LIN {X 0,Y 675.364,Z 1023.131,A -85,B 0,C 180,E1 30768.288,E2 30768.288} C_VEL
LIN {X 0,Y 672.75,Z 1029.782,A -85,B 0,C 180,E1 30767.69,E2 30767.69} C_VEL
LIN {X 0,Y 672.369,Z 1032.5,A -85,B 0,C 180,E1 30767.398,E2 30767.398} C_VEL
LIN {X 0,Y 672.252,Z 1040.855,A -85,B 0,C 180,E1 30766.32,E2 30766.32} C_VEL
LIN {X 0,Y 672.157,Z 1047.422,A -85,B 0,C 180,E1 30765.175,E2 30765.175} C_VEL
LIN {X 0,Y 672.12,Z 1051.926,A -85,B 0,C 180,E1 30764.114,E2 30764.114} C_VEL
LIN {X 0,Y 672.089,Z 1055.278,A -85,B 0,C 180,E1 30762.957,E2 30762.957} C_VEL
LIN {X 0,Y 672.074,Z 1057.172,A -85,B 0,C 180,E1 30761.615,E2 30761.615} C_VEL
LIN {X 0,Y 672.069,Z 1057.276,A -85,B 0,C 180,E1 30760.533,E2 30760.533} C_VEL
LIN {X 0,Y 672.07,Z 1056.109,A -85,B 0,C 180,E1 30759.444,E2 30759.444} C_VEL
LIN {X 0,Y 672.096,Z 1053.112,A -85,B 0,C 180,E1 30758.165,E2 30758.165} C_VEL
LIN {X 0,Y 672.133,Z 1048.387,A -85,B 0,C 180,E1 30756.968,E2 30756.968} C_VEL
LIN {X 0,Y 672.186,Z 1042.857,A -85,B 0,C 180,E1 30755.947,E2 30755.947} C_VEL
LIN {X 0,Y 672.298,Z 1034.959,A -85,B 0,C 180,E1 30754.826,E2 30754.826} C_VEL
LIN {X 0,Y 672.444,Z 1025.328,A -85,B 0,C 180,E1 30753.792,E2 30753.792} C_VEL
LIN {X 0,Y 672.579,Z 1016.19,A -85,B 0,C 180,E1 30753.012,E2 30753.012} C_VEL
LIN {X 0,Y 672.716,Z 1005.111,A -85,B 0,C 180,E1 30752.247,E2 30752.247} C_VEL
LIN {X 0,Y 672.919,Z 991.221,A -85,B 0,C 180,E1 30751.512,E2 30751.512} C_VEL
LIN {X 0,Y 673.04,Z 978.297,A -85,B 0,C 180,E1 30751.008,E2 30751.008} C_VEL
LIN {X 0,Y 673.159,Z 964.07,A -85,B 0,C 180,E1 30750.609,E2 30750.609} C_VEL
LIN {X 0,Y 673.195,Z 947.441,A -85,B 0,C 180,E1 30750.341,E2 30750.341} C_VEL
LIN {X 0,Y 673.46,Z 838.836,A -85,B 0,C 180,E1 30749.163,E2 30749.163} C_VEL
LIN {X 0,Y 674.164,Z 758.895,A -85,B 0,C 180,E1 30746.003,E2 30746.003} C_VEL
LIN {X 0,Y 674.908,Z 679.946,A -85,B 0,C 180,E1 30742.883,E2 30742.883} C_VEL
LIN {X 0,Y 675.546,Z 603.018,A -85,B 0,C 180,E1 30739.85,E2 30739.85} C_VEL
LIN {X 0,Y 676.134,Z 525.625,A -85,B 0,C 180,E1 30736.788,E2 30736.788} C_VEL
LIN {X 0,Y 676.398,Z 479.441,A -85,B 0,C 180,E1 30734.947,E2 30734.947} C_VEL
LIN {X 0,Y 677.625,Z 481.415,A -85,B 0,C 180,E1 30734.815,E2 30734.815} C_VEL
LIN {X 0,Y 679.206,Z 481.602,A -85,B 0,C 180,E1 30734.68,E2 30734.68} C_VEL
LIN {X 0,Y 681.86,Z 479.707,A -85,B 0,C 180,E1 30734.487,E2 30734.487} C_VEL
LIN {X 0,Y 685.332,Z 474.609,A -85,B 0,C 180,E1 30734.275,E2 30734.275} C_VEL
LIN {X 0,Y 686.171,Z 473.174,A -85,B 0,C 180,E1 30734.227,E2 30734.227} C_VEL
LIN {X 0,Y 689.689,Z 471.896,A -85,B 0,C 180,E1 30733.961,E2 30733.961} C_VEL
LIN {X 0,Y 693.542,Z 468.674,A -85,B 0,C 180,E1 30733.699,E2 30733.699} C_VEL
LIN {X 0,Y 691.039,Z 679.216,A -85,B 0,C 180,E1 30730.991,E2 30730.991} C_VEL
LIN {X 0,Y 689.557,Z 799.238,A -85,B 0,C 180,E1 30729.461,E2 30729.461} C_VEL
LIN {X 0,Y 688.803,Z 826.662,A -85,B 0,C 180,E1 30728.964,E2 30728.964} C_VEL
LIN {X 0,Y 687.772,Z 853.657,A -85,B 0,C 180,E1 30728.297,E2 30728.297} C_VEL
LIN {X 0,Y 686.749,Z 876.496,A -85,B 0,C 180,E1 30727.594,E2 30727.594} C_VEL
LIN {X 0,Y 685.634,Z 898.908,A -85,B 0,C 180,E1 30726.779,E2 30726.779} C_VEL
LIN {X 0,Y 684.187,Z 925.781,A -85,B 0,C 180,E1 30725.624,E2 30725.624} C_VEL
LIN {X 0,Y 682.832,Z 948.662,A -85,B 0,C 180,E1 30724.47,E2 30724.47} C_VEL
LIN {X 0,Y 681.518,Z 969.977,A -85,B 0,C 180,E1 30723.25,E2 30723.25} C_VEL
LIN {X 0,Y 679.995,Z 993.701,A -85,B 0,C 180,E1 30721.715,E2 30721.715} C_VEL
LIN {X 0,Y 678.508,Z 1017.521,A -85,B 0,C 180,E1 30719.944,E2 30719.944} C_VEL
LIN {X 0,Y 677.131,Z 1039.319,A -85,B 0,C 180,E1 30718.103,E2 30718.103} C_VEL
LIN {X 0,Y 675.956,Z 1059.69,A -85,B 0,C 180,E1 30716.156,E2 30716.156} C_VEL
LIN {X 0,Y 674.879,Z 1078.449,A -85,B 0,C 180,E1 30714.124,E2 30714.124} C_VEL
LIN {X 0,Y 674.182,Z 1092.611,A -85,B 0,C 180,E1 30712.406,E2 30712.406} C_VEL
LIN {X 0,Y 673.586,Z 1105.407,A -85,B 0,C 180,E1 30710.69,E2 30710.69} C_VEL
LIN {X 0,Y 673.039,Z 1119.756,A -85,B 0,C 180,E1 30708.538,E2 30708.538} C_VEL
LIN {X 0,Y 672.594,Z 1131.955,A -85,B 0,C 180,E1 30706.408,E2 30706.408} C_VEL
LIN {X 0,Y 672.363,Z 1141.26,A -85,B 0,C 180,E1 30704.557,E2 30704.557} C_VEL
LIN {X 0,Y 672.181,Z 1149.32,A -85,B 0,C 180,E1 30702.719,E2 30702.719} C_VEL
LIN {X 0,Y 672.03,Z 1156.847,A -85,B 0,C 180,E1 30700.719,E2 30700.719} C_VEL
LIN {X 0,Y 671.972,Z 1163.694,A -85,B 0,C 180,E1 30698.472,E2 30698.472} C_VEL
LIN {X 0,Y 671.93,Z 1169.194,A -85,B 0,C 180,E1 30696.066,E2 30696.066} C_VEL
LIN {X 0,Y 671.912,Z 1172.615,A -85,B 0,C 180,E1 30693.841,E2 30693.841} C_VEL
LIN {X 0,Y 671.907,Z 1174.487,A -85,B 0,C 180,E1 30691.707,E2 30691.707} C_VEL
LIN {X 0,Y 671.892,Z 1174.892,A -85,B 0,C 180,E1 30689.404,E2 30689.404} C_VEL
LIN {X 0,Y 671.911,Z 1173.798,A -85,B 0,C 180,E1 30687.186,E2 30687.186} C_VEL
LIN {X 0,Y 671.921,Z 1170.978,A -85,B 0,C 180,E1 30684.879,E2 30684.879} C_VEL
LIN {X 0,Y 671.942,Z 1166.841,A -85,B 0,C 180,E1 30682.735,E2 30682.735} C_VEL
LIN {X 0,Y 671.993,Z 1161.255,A -85,B 0,C 180,E1 30680.58,E2 30680.58} C_VEL
LIN {X 0,Y 672.098,Z 1153.81,A -85,B 0,C 180,E1 30678.328,E2 30678.328} C_VEL
LIN {X 0,Y 672.281,Z 1143.661,A -85,B 0,C 180,E1 30675.867,E2 30675.867} C_VEL
LIN {X 0,Y 672.539,Z 1134.3,A -85,B 0,C 180,E1 30673.948,E2 30673.948} C_VEL
LIN {X 0,Y 672.826,Z 1124.996,A -85,B 0,C 180,E1 30672.264,E2 30672.264} C_VEL
LIN {X 0,Y 673.218,Z 1114.542,A -85,B 0,C 180,E1 30670.569,E2 30670.569} C_VEL
LIN {X 0,Y 673.702,Z 1102.836,A -85,B 0,C 180,E1 30668.861,E2 30668.861} C_VEL
LIN {X 0,Y 674.384,Z 1088.32,A -85,B 0,C 180,E1 30666.958,E2 30666.958} C_VEL
LIN {X 0,Y 675.338,Z 1070.129,A -85,B 0,C 180,E1 30664.856,E2 30664.856} C_VEL
LIN {X 0,Y 676.323,Z 1052.716,A -85,B 0,C 180,E1 30663.061,E2 30663.061} C_VEL
LIN {X 0,Y 677.637,Z 1031.306,A -85,B 0,C 180,E1 30661.104,E2 30661.104} C_VEL
LIN {X 0,Y 679.06,Z 1008.592,A -85,B 0,C 180,E1 30659.275,E2 30659.275} C_VEL
LIN {X 0,Y 680.528,Z 985.671,A -85,B 0,C 180,E1 30657.655,E2 30657.655} C_VEL
LIN {X 0,Y 681.887,Z 963.817,A -85,B 0,C 180,E1 30656.29,E2 30656.29} C_VEL
LIN {X 0,Y 683.437,Z 938.443,A -85,B 0,C 180,E1 30654.904,E2 30654.904} C_VEL
LIN {X 0,Y 684.732,Z 916.065,A -85,B 0,C 180,E1 30653.849,E2 30653.849} C_VEL
LIN {X 0,Y 685.857,Z 895.012,A -85,B 0,C 180,E1 30652.982,E2 30652.982} C_VEL
LIN {X 0,Y 686.929,Z 872.513,A -85,B 0,C 180,E1 30652.183,E2 30652.183} C_VEL
LIN {X 0,Y 688.111,Z 845.903,A -85,B 0,C 180,E1 30651.4,E2 30651.4} C_VEL
LIN {X 0,Y 689.019,Z 819.031,A -85,B 0,C 180,E1 30650.793,E2 30650.793} C_VEL
LIN {X 0,Y 689.636,Z 795.197,A -85,B 0,C 180,E1 30650.39,E2 30650.39} C_VEL
LIN {X 0,Y 692.298,Z 572.503,A -85,B 0,C 180,E1 30647.558,E2 30647.558} C_VEL
LIN {X 0,Y 694.922,Z 360.278,A -85,B 0,C 180,E1 30644.783,E2 30644.783} C_VEL
LIN {X 0,Y 694.84,Z 353.662,A -85,B 0,C 180,E1 30644.681,E2 30644.681} C_VEL
LIN {X 0,Y 681.845,Z 334.472,A -85,B 0,C 180,E1 30643.28,E2 30643.28} C_VEL
LIN {X 0,Y 678.625,Z 330.159,A -85,B 0,C 180,E1 30642.926,E2 30642.926} C_VEL
LIN {X 0,Y 675.796,Z 325.922,A -85,B 0,C 180,E1 30642.603,E2 30642.603} C_VEL
LIN {X 0,Y 673.561,Z 323.434,A -85,B 0,C 180,E1 30642.333,E2 30642.333} C_VEL
LIN {X 0,Y 672.581,Z 320.456,A -85,B 0,C 180,E1 30641.806,E2 30641.806} C_VEL
LIN {X 0,Y 672.563,Z 320.456,A -85,B 0,C 180,E1 30638.832,E2 30638.832} C_VEL
LIN {X 0,Y 672.571,Z 320.453,A -85,B 0,C 180,E1 30635.856,E2 30635.856} C_VEL
LIN {X 0,Y 672.556,Z 320.433,A -85,B 0,C 180,E1 30632.864,E2 30632.864} C_VEL
LIN {X 0,Y 672.574,Z 320.431,A -85,B 0,C 180,E1 30629.924,E2 30629.924} C_VEL
LIN {X 0,Y 672.571,Z 320.455,A -85,B 0,C 180,E1 30626.869,E2 30626.869} C_VEL
LIN {X 0,Y 672.582,Z 320.437,A -85,B 0,C 180,E1 30623.852,E2 30623.852} C_VEL
LIN {X 0,Y 672.582,Z 320.429,A -85,B 0,C 180,E1 30620.63,E2 30620.63} C_VEL
LIN {X 0,Y 672.563,Z 320.456,A -85,B 0,C 180,E1 30617.649,E2 30617.649} C_VEL
LIN {X 0,Y 672.586,Z 320.437,A -85,B 0,C 180,E1 30614.551,E2 30614.551} C_VEL
LIN {X 0,Y 672.554,Z 320.436,A -85,B 0,C 180,E1 30611.563,E2 30611.563} C_VEL
LIN {X 0,Y 672.575,Z 320.456,A -85,B 0,C 180,E1 30608.55,E2 30608.55} C_VEL
LIN {X 0,Y 672.559,Z 320.433,A -85,B 0,C 180,E1 30605.545,E2 30605.545} C_VEL
LIN {X 0,Y 672.585,Z 320.437,A -85,B 0,C 180,E1 30602.556,E2 30602.556} C_VEL
LIN {X 0,Y 672.588,Z 320.454,A -85,B 0,C 180,E1 30599.319,E2 30599.319} C_VEL
LIN {X 0,Y 672.585,Z 320.441,A -85,B 0,C 180,E1 30596.079,E2 30596.079} C_VEL
LIN {X 0,Y 672.561,Z 320.426,A -85,B 0,C 180,E1 30593.169,E2 30593.169} C_VEL
LIN {X 0,Y 672.588,Z 320.433,A -85,B 0,C 180,E1 30590.07,E2 30590.07} C_VEL
LIN {X 0,Y 672.556,Z 320.452,A -85,B 0,C 180,E1 30587.027,E2 30587.027} C_VEL
LIN {X 0,Y 672.602,Z 320.598,A -85,B 0,C 180,E1 30586.503,E2 30586.503} C_VEL
LIN {X 0,Y 673.919,Z 323.961,A -85,B 0,C 180,E1 30585.917,E2 30585.917} C_VEL
LIN {X 0,Y 675.538,Z 326.131,A -85,B 0,C 180,E1 30585.426,E2 30585.426} C_VEL
LIN {X 0,Y 677.325,Z 329.76,A -85,B 0,C 180,E1 30584.765,E2 30584.765} C_VEL
LIN {X 0,Y 678.38,Z 331.366,A -85,B 0,C 180,E1 30584.439,E2 30584.439} C_VEL
LIN {X 0,Y 680.601,Z 335.361,A -85,B 0,C 180,E1 30583.704,E2 30583.704} C_VEL
LIN {X 0,Y 686.363,Z 346.276,A -85,B 0,C 180,E1 30581.835,E2 30581.835} C_VEL
LIN {X 0,Y 693.008,Z 358.872,A -85,B 0,C 180,E1 30579.828,E2 30579.828} C_VEL
LIN {X 0,Y 695.642,Z 364.353,A -85,B 0,C 180,E1 30579.028,E2 30579.028} C_VEL
LIN {X 0,Y 693.695,Z 398.694,A -85,B 0,C 180,E1 30576.332,E2 30576.332} C_VEL
LIN {X 0,Y 691.737,Z 435.157,A -85,B 0,C 180,E1 30573.614,E2 30573.614} C_VEL
LIN {X 0,Y 689.802,Z 473.923,A -85,B 0,C 180,E1 30570.853,E2 30570.853} C_VEL
LIN {X 0,Y 687.855,Z 515.666,A -85,B 0,C 180,E1 30568.004,E2 30568.004} C_VEL
LIN {X 0,Y 686.907,Z 547.596,A -85,B 0,C 180,E1 30565.864,E2 30565.864} C_VEL
LIN {X 0,Y 688.183,Z 560.103,A -85,B 0,C 180,E1 30564.925,E2 30564.925} C_VEL
LIN {X 0,Y 691.006,Z 570.711,A -85,B 0,C 180,E1 30564.021,E2 30564.021} C_VEL
LIN {X 0,Y 695.237,Z 579.657,A -85,B 0,C 180,E1 30563.149,E2 30563.149} C_VEL
LIN {X 0,Y 700.518,Z 586.818,A -85,B 0,C 180,E1 30562.344,E2 30562.344} C_VEL
LIN {X 0,Y 707.26,Z 592.952,A -85,B 0,C 180,E1 30561.534,E2 30561.534} C_VEL
LIN {X 0,Y 715.53,Z 597.88,A -85,B 0,C 180,E1 30560.726,E2 30560.726} C_VEL
LIN {X 0,Y 719.508,Z 599.149,A -85,B 0,C 180,E1 30560.263,E2 30560.263} C_VEL
LIN {X 0,Y 722.076,Z 599.031,A -85,B 0,C 180,E1 30559.812,E2 30559.812} C_VEL
LIN {X 0,Y 723.653,Z 597.658,A -85,B 0,C 180,E1 30559.294,E2 30559.294} C_VEL
LIN {X 0,Y 723.84,Z 595.33,A -85,B 0,C 180,E1 30558.835,E2 30558.835} C_VEL
LIN {X 0,Y 722.65,Z 591.882,A -85,B 0,C 180,E1 30558.383,E2 30558.383} C_VEL
LIN {X 0,Y 720.082,Z 587.576,A -85,B 0,C 180,E1 30558.005,E2 30558.005} C_VEL
LIN {X 0,Y 713.477,Z 578.261,A -85,B 0,C 180,E1 30557.502,E2 30557.502} C_VEL
LIN {X 0,Y 707.234,Z 566.846,A -85,B 0,C 180,E1 30557.037,E2 30557.037} C_VEL
LIN {X 0,Y 702.128,Z 554.061,A -85,B 0,C 180,E1 30556.648,E2 30556.648} C_VEL
LIN {X 0,Y 698.275,Z 540.169,A -85,B 0,C 180,E1 30556.348,E2 30556.348} C_VEL
LIN {X 0,Y 695.658,Z 524.951,A -85,B 0,C 180,E1 30556.142,E2 30556.142} C_VEL
LIN {X 0,Y 694.307,Z 508.233,A -85,B 0,C 180,E1 30556.035,E2 30556.035} C_VEL
LIN {X 0,Y 694.082,Z 360.627,A -85,B 0,C 180,E1 30556.017,E2 30556.017} C_VEL
LIN {X 0,Y 692.049,Z 361.517,A -85,B 0,C 180,E1 30555.854,E2 30555.854} C_VEL
LIN {X 0,Y 695.128,Z 375.054,A -85,B 0,C 180,E1 30555.373,E2 30555.373} C_VEL
LIN {X 0,Y 692.51,Z 584.112,A -85,B 0,C 180,E1 30552.635,E2 30552.635} C_VEL
LIN {X 0,Y 689.944,Z 807.11,A -85,B 0,C 180,E1 30549.804,E2 30549.804} C_VEL
LIN {X 0,Y 689.372,Z 837.488,A -85,B 0,C 180,E1 30549.377,E2 30549.377} C_VEL
LIN {X 0,Y 688.527,Z 864.544,A -85,B 0,C 180,E1 30548.833,E2 30548.833} C_VEL
LIN {X 0,Y 687.488,Z 890.496,A -85,B 0,C 180,E1 30548.148,E2 30548.148} C_VEL
LIN {X 0,Y 686.237,Z 918.163,A -85,B 0,C 180,E1 30547.233,E2 30547.233} C_VEL
LIN {X 0,Y 684.993,Z 941.728,A -85,B 0,C 180,E1 30546.296,E2 30546.296} C_VEL
LIN {X 0,Y 683.77,Z 963.074,A -85,B 0,C 180,E1 30545.316,E2 30545.316} C_VEL
LIN {X 0,Y 682.296,Z 987.342,A -85,B 0,C 180,E1 30544.041,E2 30544.041} C_VEL
LIN {X 0,Y 680.793,Z 1010.836,A -85,B 0,C 180,E1 30542.615,E2 30542.615} C_VEL
LIN {X 0,Y 679.515,Z 1031.617,A -85,B 0,C 180,E1 30541.194,E2 30541.194} C_VEL
LIN {X 0,Y 678.045,Z 1054.695,A -85,B 0,C 180,E1 30539.409,E2 30539.409} C_VEL
LIN {X 0,Y 676.801,Z 1074.892,A -85,B 0,C 180,E1 30537.637,E2 30537.637} C_VEL
LIN {X 0,Y 675.589,Z 1095.443,A -85,B 0,C 180,E1 30535.604,E2 30535.604} C_VEL
LIN {X 0,Y 674.749,Z 1111.068,A -85,B 0,C 180,E1 30533.861,E2 30533.861} C_VEL
LIN {X 0,Y 674.014,Z 1126.16,A -85,B 0,C 180,E1 30532,E2 30532} C_VEL
LIN {X 0,Y 673.323,Z 1141.967,A -85,B 0,C 180,E1 30529.789,E2 30529.789} C_VEL
LIN {X 0,Y 672.843,Z 1154.882,A -85,B 0,C 180,E1 30527.716,E2 30527.716} C_VEL
LIN {X 0,Y 672.498,Z 1165.947,A -85,B 0,C 180,E1 30525.699,E2 30525.699} C_VEL
LIN {X 0,Y 672.228,Z 1177.033,A -85,B 0,C 180,E1 30523.328,E2 30523.328} C_VEL
LIN {X 0,Y 672.048,Z 1185.838,A -85,B 0,C 180,E1 30521.064,E2 30521.064} C_VEL
LIN {X 0,Y 671.973,Z 1193.113,A -85,B 0,C 180,E1 30518.729,E2 30518.729} C_VEL
LIN {X 0,Y 671.933,Z 1198.43,A -85,B 0,C 180,E1 30516.493,E2 30516.493} C_VEL
LIN {X 0,Y 671.919,Z 1202.166,A -85,B 0,C 180,E1 30514.266,E2 30514.266} C_VEL
LIN {X 0,Y 671.91,Z 1204.376,A -85,B 0,C 180,E1 30511.96,E2 30511.96} C_VEL
LIN {X 0,Y 671.892,Z 1204.915,A -85,B 0,C 180,E1 30509.573,E2 30509.573} C_VEL
LIN {X 0,Y 671.908,Z 1203.983,A -85,B 0,C 180,E1 30507.44,E2 30507.44} C_VEL
LIN {X 0,Y 671.918,Z 1201.293,A -85,B 0,C 180,E1 30505.133,E2 30505.133} C_VEL
LIN {X 0,Y 671.941,Z 1197.139,A -85,B 0,C 180,E1 30502.904,E2 30502.904} C_VEL
LIN {X 0,Y 671.992,Z 1191.407,A -85,B 0,C 180,E1 30500.665,E2 30500.665} C_VEL
LIN {X 0,Y 672.094,Z 1183.956,A -85,B 0,C 180,E1 30498.413,E2 30498.413} C_VEL
LIN {X 0,Y 672.289,Z 1173.964,A -85,B 0,C 180,E1 30495.969,E2 30495.969} C_VEL
LIN {X 0,Y 672.553,Z 1163.609,A -85,B 0,C 180,E1 30493.857,E2 30493.857} C_VEL
LIN {X 0,Y 672.924,Z 1152.668,A -85,B 0,C 180,E1 30491.907,E2 30491.907} C_VEL
LIN {X 0,Y 673.499,Z 1138.333,A -85,B 0,C 180,E1 30489.671,E2 30489.671} C_VEL
LIN {X 0,Y 674.166,Z 1122.97,A -85,B 0,C 180,E1 30487.593,E2 30487.593} C_VEL
LIN {X 0,Y 674.859,Z 1108.709,A -85,B 0,C 180,E1 30485.862,E2 30485.862} C_VEL
LIN {X 0,Y 675.939,Z 1089.794,A -85,B 0,C 180,E1 30483.812,E2 30483.812} C_VEL
LIN {X 0,Y 676.993,Z 1071.309,A -85,B 0,C 180,E1 30482.034,E2 30482.034} C_VEL
LIN {X 0,Y 678.354,Z 1050.054,A -85,B 0,C 180,E1 30480.215,E2 30480.215} C_VEL
LIN {X 0,Y 679.666,Z 1028.935,A -85,B 0,C 180,E1 30478.614,E2 30478.614} C_VEL
LIN {X 0,Y 681.041,Z 1007.088,A -85,B 0,C 180,E1 30477.141,E2 30477.141} C_VEL
LIN {X 0,Y 682.637,Z 982.152,A -85,B 0,C 180,E1 30475.672,E2 30475.672} C_VEL
LIN {X 0,Y 683.966,Z 959.602,A -85,B 0,C 180,E1 30474.517,E2 30474.517} C_VEL
LIN {X 0,Y 685.296,Z 936.194,A -85,B 0,C 180,E1 30473.466,E2 30473.466} C_VEL
LIN {X 0,Y 686.637,Z 909.294,A -85,B 0,C 180,E1 30472.451,E2 30472.451} C_VEL
LIN {X 0,Y 687.792,Z 883.751,A -85,B 0,C 180,E1 30471.658,E2 30471.658} C_VEL
LIN {X 0,Y 688.756,Z 857.273,A -85,B 0,C 180,E1 30471.006,E2 30471.006} C_VEL
LIN {X 0,Y 689.538,Z 830.262,A -85,B 0,C 180,E1 30470.508,E2 30470.508} C_VEL
LIN {X 0,Y 690.628,Z 745.888,A -85,B 0,C 180,E1 30469.428,E2 30469.428} C_VEL
LIN {X 0,Y 693.249,Z 523.728,A -85,B 0,C 180,E1 30466.584,E2 30466.584} C_VEL
LIN {X 0,Y 695.286,Z 354.322,A -85,B 0,C 180,E1 30464.34,E2 30464.34} C_VEL
LIN {X 0,Y 693.021,Z 350.722,A -85,B 0,C 180,E1 30464.068,E2 30464.068} C_VEL
LIN {X 0,Y 695.397,Z 350.142,A -85,B 0,C 180,E1 30463.873,E2 30463.873} C_VEL
LIN {X 0,Y 697.141,Z 348.137,A -85,B 0,C 180,E1 30463.707,E2 30463.707} C_VEL
LIN {X 0,Y 700.205,Z 350.666,A -85,B 0,C 180,E1 30463.257,E2 30463.257} C_VEL
LIN {X 0,Y 701.743,Z 352.07,A -85,B 0,C 180,E1 30462.793,E2 30462.793} C_VEL
LIN {X 0,Y 701.941,Z 352.679,A -85,B 0,C 180,E1 30462.249,E2 30462.249} C_VEL
LIN {X 0,Y 700.564,Z 352.305,A -85,B 0,C 180,E1 30461.715,E2 30461.715} C_VEL
LIN {X 0,Y 697.833,Z 350.943,A -85,B 0,C 180,E1 30461.232,E2 30461.232} C_VEL
LIN {X 0,Y 693.066,Z 347.654,A -85,B 0,C 180,E1 30460.701,E2 30460.701} C_VEL
LIN {X 0,Y 685.428,Z 339.878,A -85,B 0,C 180,E1 30459.822,E2 30459.822} C_VEL
LIN {X 0,Y 682.392,Z 335.579,A -85,B 0,C 180,E1 30459.435,E2 30459.435} C_VEL
LIN {X 0,Y 679.119,Z 330.875,A -85,B 0,C 180,E1 30459.008,E2 30459.008} C_VEL
LIN {X 0,Y 676.5,Z 326.967,A -85,B 0,C 180,E1 30458.657,E2 30458.657} C_VEL
LIN {X 0,Y 675.471,Z 325.664,A -85,B 0,C 180,E1 30458.523,E2 30458.523} C_VEL
LIN {X 0,Y 673.205,Z 322.716,A -85,B 0,C 180,E1 30458.225,E2 30458.225} C_VEL
LIN {X 0,Y 672.57,Z 320.44,A -85,B 0,C 180,E1 30458.095,E2 30458.095} C_VEL
LIN {X 0,Y 672.582,Z 320.439,A -85,B 0,C 180,E1 30455.019,E2 30455.019} C_VEL
LIN {X 0,Y 672.553,Z 320.42,A -85,B 0,C 180,E1 30451.956,E2 30451.956} C_VEL
LIN {X 0,Y 672.555,Z 320.456,A -85,B 0,C 180,E1 30449.051,E2 30449.051} C_VEL
LIN {X 0,Y 672.582,Z 320.413,A -85,B 0,C 180,E1 30446.107,E2 30446.107} C_VEL
LIN {X 0,Y 672.557,Z 320.455,A -85,B 0,C 180,E1 30443.11,E2 30443.11} C_VEL
LIN {X 0,Y 672.591,Z 320.445,A -85,B 0,C 180,E1 30439.904,E2 30439.904} C_VEL
LIN {X 0,Y 672.574,Z 320.446,A -85,B 0,C 180,E1 30436.852,E2 30436.852} C_VEL
LIN {X 0,Y 672.584,Z 320.452,A -85,B 0,C 180,E1 30433.673,E2 30433.673} C_VEL
LIN {X 0,Y 672.581,Z 320.574,A -85,B 0,C 180,E1 30432.133,E2 30432.133} C_VEL
LIN {X 0,Y 674.534,Z 328.275,A -85,B 0,C 180,E1 30431.826,E2 30431.826} C_VEL
LIN {X 0,Y 674.597,Z 404.567,A -85,B 0,C 180,E1 30429.211,E2 30429.211} C_VEL
LIN {X 0,Y 675.029,Z 489.424,A -85,B 0,C 180,E1 30426.165,E2 30426.165} C_VEL
LIN {X 0,Y 675.207,Z 555.997,A -85,B 0,C 180,E1 30423.693,E2 30423.693} C_VEL
LIN {X 0,Y 675.047,Z 618.673,A -85,B 0,C 180,E1 30421.316,E2 30421.316} C_VEL
LIN {X 0,Y 674.608,Z 698.374,A -85,B 0,C 180,E1 30418.259,E2 30418.259} C_VEL
LIN {X 0,Y 674.047,Z 772.814,A -85,B 0,C 180,E1 30415.363,E2 30415.363} C_VEL
LIN {X 0,Y 673.48,Z 841.27,A -85,B 0,C 180,E1 30412.698,E2 30412.698} C_VEL
LIN {X 0,Y 673.176,Z 955.75,A -85,B 0,C 180,E1 30411.453,E2 30411.453} C_VEL
LIN {X 0,Y 673.114,Z 968.927,A -85,B 0,C 180,E1 30411.183,E2 30411.183} C_VEL
LIN {X 0,Y 673.031,Z 981.267,A -85,B 0,C 180,E1 30410.81,E2 30410.81} C_VEL
LIN {X 0,Y 672.891,Z 995.65,A -85,B 0,C 180,E1 30410.204,E2 30410.204} C_VEL
LIN {X 0,Y 672.726,Z 1007.164,A -85,B 0,C 180,E1 30409.553,E2 30409.553} C_VEL
LIN {X 0,Y 672.602,Z 1017.596,A -85,B 0,C 180,E1 30408.814,E2 30408.814} C_VEL
LIN {X 0,Y 672.444,Z 1027.912,A -85,B 0,C 180,E1 30407.898,E2 30407.898} C_VEL
LIN {X 0,Y 672.369,Z 1032.5,A -85,B 0,C 180,E1 30407.398,E2 30407.398} C_VEL
LIN {X 0,Y 671.338,Z 1037.095,A -85,B 0,C 180,E1 30406.872,E2 30406.872} C_VEL
LIN {X 0,Y 666.831,Z 1044.621,A -85,B 0,C 180,E1 30405.874,E2 30405.874} C_VEL
LIN {X 0,Y 664.609,Z 1048.549,A -85,B 0,C 180,E1 30405.211,E2 30405.211} C_VEL
LIN {X 0,Y 664.239,Z 1050.248,A -85,B 0,C 180,E1 30404.861,E2 30404.861} C_VEL
LIN {X 0,Y 664.179,Z 1055.004,A -85,B 0,C 180,E1 30403.532,E2 30403.532} C_VEL
LIN {X 0,Y 664.158,Z 1057.291,A -85,B 0,C 180,E1 30402.476,E2 30402.476} C_VEL
LIN {X 0,Y 664.148,Z 1058.349,A -85,B 0,C 180,E1 30401.478,E2 30401.478} C_VEL
LIN {X 0,Y 664.145,Z 1058.338,A -85,B 0,C 180,E1 30400.47,E2 30400.47} C_VEL
LIN {X 0,Y 664.144,Z 1057.103,A -85,B 0,C 180,E1 30399.372,E2 30399.372} C_VEL
LIN {X 0,Y 664.179,Z 1053.995,A -85,B 0,C 180,E1 30398.077,E2 30398.077} C_VEL
LIN {X 0,Y 664.219,Z 1049.138,A -85,B 0,C 180,E1 30396.865,E2 30396.865} C_VEL
LIN {X 0,Y 664.28,Z 1043.501,A -85,B 0,C 180,E1 30395.831,E2 30395.831} C_VEL
LIN {X 0,Y 664.402,Z 1035.913,A -85,B 0,C 180,E1 30394.753,E2 30394.753} C_VEL
LIN {X 0,Y 664.551,Z 1026.499,A -85,B 0,C 180,E1 30393.734,E2 30393.734} C_VEL
LIN {X 0,Y 664.696,Z 1017.328,A -85,B 0,C 180,E1 30392.941,E2 30392.941} C_VEL
LIN {X 0,Y 664.823,Z 1007.477,A -85,B 0,C 180,E1 30392.246,E2 30392.246} C_VEL
LIN {X 0,Y 664.993,Z 996.032,A -85,B 0,C 180,E1 30391.596,E2 30391.596} C_VEL
LIN {X 0,Y 665.147,Z 982.055,A -85,B 0,C 180,E1 30391,E2 30391} C_VEL
LIN {X 0,Y 665.242,Z 969.419,A -85,B 0,C 180,E1 30390.613,E2 30390.613} C_VEL
LIN {X 0,Y 665.298,Z 956.949,A -85,B 0,C 180,E1 30390.352,E2 30390.352} C_VEL
LIN {X 0,Y 665.374,Z 928.558,A -85,B 0,C 180,E1 30390.018,E2 30390.018} C_VEL
LIN {X 0,Y 665.649,Z 839.963,A -85,B 0,C 180,E1 30389.042,E2 30389.042} C_VEL
LIN {X 0,Y 666.415,Z 758.532,A -85,B 0,C 180,E1 30385.805,E2 30385.805} C_VEL
LIN {X 0,Y 667.184,Z 680.601,A -85,B 0,C 180,E1 30382.713,E2 30382.713} C_VEL
LIN {X 0,Y 667.883,Z 603.228,A -85,B 0,C 180,E1 30379.644,E2 30379.644} C_VEL
LIN {X 0,Y 668.568,Z 526.073,A -85,B 0,C 180,E1 30376.563,E2 30376.563} C_VEL
LIN {X 0,Y 668.78,Z 495.929,A -85,B 0,C 180,E1 30375.356,E2 30375.356} C_VEL
LIN {X 0,Y 670.012,Z 497.917,A -85,B 0,C 180,E1 30375.22,E2 30375.22} C_VEL
LIN {X 0,Y 671.766,Z 498.007,A -85,B 0,C 180,E1 30375.068,E2 30375.068} C_VEL
LIN {X 0,Y 674.525,Z 495.749,A -85,B 0,C 180,E1 30374.866,E2 30374.866} C_VEL
LIN {X 0,Y 678.117,Z 490.099,A -85,B 0,C 180,E1 30374.647,E2 30374.647} C_VEL
LIN {X 0,Y 678.518,Z 489.577,A -85,B 0,C 180,E1 30374.621,E2 30374.621} C_VEL
LIN {X 0,Y 682.012,Z 488.319,A -85,B 0,C 180,E1 30374.35,E2 30374.35} C_VEL
LIN {X 0,Y 685.894,Z 484.798,A -85,B 0,C 180,E1 30374.083,E2 30374.083} C_VEL
LIN {X 0,Y 687.579,Z 482.678,A -85,B 0,C 180,E1 30373.977,E2 30373.977} C_VEL
LIN {X 0,Y 684.728,Z 701.394,A -85,B 0,C 180,E1 30371.149,E2 30371.149} C_VEL
LIN {X 0,Y 683.371,Z 799.352,A -85,B 0,C 180,E1 30369.888,E2 30369.888} C_VEL
LIN {X 0,Y 682.543,Z 826.828,A -85,B 0,C 180,E1 30369.387,E2 30369.387} C_VEL
LIN {X 0,Y 681.418,Z 853.767,A -85,B 0,C 180,E1 30368.717,E2 30368.717} C_VEL
LIN {X 0,Y 680.309,Z 876.507,A -85,B 0,C 180,E1 30368.013,E2 30368.013} C_VEL
LIN {X 0,Y 679.168,Z 897.796,A -85,B 0,C 180,E1 30367.236,E2 30367.236} C_VEL
LIN {X 0,Y 677.721,Z 922.342,A -85,B 0,C 180,E1 30366.193,E2 30366.193} C_VEL
LIN {X 0,Y 676.065,Z 947.796,A -85,B 0,C 180,E1 30364.916,E2 30364.916} C_VEL
LIN {X 0,Y 674.599,Z 969.53,A -85,B 0,C 180,E1 30363.666,E2 30363.666} C_VEL
LIN {X 0,Y 672.944,Z 993.254,A -85,B 0,C 180,E1 30362.12,E2 30362.12} C_VEL
LIN {X 0,Y 671.266,Z 1017.18,A -85,B 0,C 180,E1 30360.329,E2 30360.329} C_VEL
LIN {X 0,Y 669.747,Z 1039.373,A -85,B 0,C 180,E1 30358.437,E2 30358.437} C_VEL
LIN {X 0,Y 668.388,Z 1060.206,A -85,B 0,C 180,E1 30356.423,E2 30356.423} C_VEL
LIN {X 0,Y 667.245,Z 1078.337,A -85,B 0,C 180,E1 30354.432,E2 30354.432} C_VEL
LIN {X 0,Y 666.447,Z 1092.663,A -85,B 0,C 180,E1 30352.675,E2 30352.675} C_VEL
LIN {X 0,Y 665.761,Z 1106.056,A -85,B 0,C 180,E1 30350.852,E2 30350.852} C_VEL
LIN {X 0,Y 665.125,Z 1120.807,A -85,B 0,C 180,E1 30348.585,E2 30348.585} C_VEL
LIN {X 0,Y 664.666,Z 1132.423,A -85,B 0,C 180,E1 30346.519,E2 30346.519} C_VEL
LIN {X 0,Y 664.407,Z 1141.674,A -85,B 0,C 180,E1 30344.646,E2 30344.646} C_VEL
LIN {X 0,Y 664.208,Z 1149.68,A -85,B 0,C 180,E1 30342.786,E2 30342.786} C_VEL
LIN {X 0,Y 664.041,Z 1157.435,A -85,B 0,C 180,E1 30340.674,E2 30340.674} C_VEL
LIN {X 0,Y 663.975,Z 1164.146,A -85,B 0,C 180,E1 30338.4,E2 30338.4} C_VEL
LIN {X 0,Y 663.929,Z 1169.491,A -85,B 0,C 180,E1 30335.966,E2 30335.966} C_VEL
LIN {X 0,Y 663.912,Z 1172.716,A -85,B 0,C 180,E1 30333.801,E2 30333.801} C_VEL
LIN {X 0,Y 663.907,Z 1174.533,A -85,B 0,C 180,E1 30331.641,E2 30331.641} C_VEL
LIN {X 0,Y 663.892,Z 1174.895,A -85,B 0,C 180,E1 30329.397,E2 30329.397} C_VEL
LIN {X 0,Y 663.912,Z 1173.798,A -85,B 0,C 180,E1 30327.152,E2 30327.152} C_VEL
LIN {X 0,Y 663.921,Z 1170.974,A -85,B 0,C 180,E1 30324.817,E2 30324.817} C_VEL
LIN {X 0,Y 663.944,Z 1166.837,A -85,B 0,C 180,E1 30322.647,E2 30322.647} C_VEL
LIN {X 0,Y 664.001,Z 1161.253,A -85,B 0,C 180,E1 30320.467,E2 30320.467} C_VEL
LIN {X 0,Y 664.116,Z 1153.809,A -85,B 0,C 180,E1 30318.186,E2 30318.186} C_VEL
LIN {X 0,Y 664.336,Z 1143.733,A -85,B 0,C 180,E1 30315.711,E2 30315.711} C_VEL
LIN {X 0,Y 664.61,Z 1134.297,A -85,B 0,C 180,E1 30313.751,E2 30313.751} C_VEL
LIN {X 0,Y 664.948,Z 1124.992,A -85,B 0,C 180,E1 30312.047,E2 30312.047} C_VEL
LIN {X 0,Y 665.373,Z 1114.539,A -85,B 0,C 180,E1 30310.331,E2 30310.331} C_VEL
LIN {X 0,Y 665.934,Z 1102.673,A -85,B 0,C 180,E1 30308.58,E2 30308.58} C_VEL
LIN {X 0,Y 666.783,Z 1086.877,A -85,B 0,C 180,E1 30306.493,E2 30306.493} C_VEL
LIN {X 0,Y 667.772,Z 1069.272,A -85,B 0,C 180,E1 30304.456,E2 30304.456} C_VEL
LIN {X 0,Y 668.893,Z 1052.176,A -85,B 0,C 180,E1 30302.684,E2 30302.684} C_VEL
LIN {X 0,Y 670.271,Z 1031.492,A -85,B 0,C 180,E1 30300.773,E2 30300.773} C_VEL
LIN {X 0,Y 671.876,Z 1008.577,A -85,B 0,C 180,E1 30298.91,E2 30298.91} C_VEL
LIN {X 0,Y 673.459,Z 985.866,A -85,B 0,C 180,E1 30297.289,E2 30297.289} C_VEL
LIN {X 0,Y 675.021,Z 963.009,A -85,B 0,C 180,E1 30295.849,E2 30295.849} C_VEL
LIN {X 0,Y 676.757,Z 937.454,A -85,B 0,C 180,E1 30294.454,E2 30294.454} C_VEL
LIN {X 0,Y 678.109,Z 916.044,A -85,B 0,C 180,E1 30293.439,E2 30293.439} C_VEL
LIN {X 0,Y 679.298,Z 895.674,A -85,B 0,C 180,E1 30292.592,E2 30292.592} C_VEL
LIN {X 0,Y 680.431,Z 874.034,A -85,B 0,C 180,E1 30291.813,E2 30291.813} C_VEL
LIN {X 0,Y 681.658,Z 848.814,A -85,B 0,C 180,E1 30291.054,E2 30291.054} C_VEL
LIN {X 0,Y 682.736,Z 820.879,A -85,B 0,C 180,E1 30290.402,E2 30290.402} C_VEL
LIN {X 0,Y 683.43,Z 796.503,A -85,B 0,C 180,E1 30289.98,E2 30289.98} C_VEL
LIN {X 0,Y 686.319,Z 577.564,A -85,B 0,C 180,E1 30287.171,E2 30287.171} C_VEL
LIN {X 0,Y 689.222,Z 364.098,A -85,B 0,C 180,E1 30284.361,E2 30284.361} C_VEL
LIN {X 0,Y 689.156,Z 357.421,A -85,B 0,C 180,E1 30284.257,E2 30284.257} C_VEL
LIN {X 0,Y 675.762,Z 337.574,A -85,B 0,C 180,E1 30282.778,E2 30282.778} C_VEL
LIN {X 0,Y 672.377,Z 332.908,A -85,B 0,C 180,E1 30282.393,E2 30282.393} C_VEL
LIN {X 0,Y 667.679,Z 327.561,A -85,B 0,C 180,E1 30281.849,E2 30281.849} C_VEL
LIN {X 0,Y 667.079,Z 326.252,A -85,B 0,C 180,E1 30281.589,E2 30281.589} C_VEL
LIN {X 0,Y 665.012,Z 323.114,A -85,B 0,C 180,E1 30280.848,E2 30280.848} C_VEL
LIN {X 0,Y 664.633,Z 321.446,A -85,B 0,C 180,E1 30280.535,E2 30280.535} C_VEL
LIN {X 0,Y 664.649,Z 321.443,A -85,B 0,C 180,E1 30277.429,E2 30277.429} C_VEL
LIN {X 0,Y 664.635,Z 321.421,A -85,B 0,C 180,E1 30274.321,E2 30274.321} C_VEL
LIN {X 0,Y 664.653,Z 321.441,A -85,B 0,C 180,E1 30271.065,E2 30271.065} C_VEL
LIN {X 0,Y 664.616,Z 321.43,A -85,B 0,C 180,E1 30268.093,E2 30268.093} C_VEL
LIN {X 0,Y 664.642,Z 321.414,A -85,B 0,C 180,E1 30265.093,E2 30265.093} C_VEL
LIN {X 0,Y 664.619,Z 321.446,A -85,B 0,C 180,E1 30262.072,E2 30262.072} C_VEL
LIN {X 0,Y 664.648,Z 321.427,A -85,B 0,C 180,E1 30259.054,E2 30259.054} C_VEL
LIN {X 0,Y 664.633,Z 321.415,A -85,B 0,C 180,E1 30255.891,E2 30255.891} C_VEL
LIN {X 0,Y 664.649,Z 321.441,A -85,B 0,C 180,E1 30252.776,E2 30252.776} C_VEL
LIN {X 0,Y 664.633,Z 321.427,A -85,B 0,C 180,E1 30249.7,E2 30249.7} C_VEL
LIN {X 0,Y 664.649,Z 321.412,A -85,B 0,C 180,E1 30246.478,E2 30246.478} C_VEL
LIN {X 0,Y 664.618,Z 321.444,A -85,B 0,C 180,E1 30243.45,E2 30243.45} C_VEL
LIN {X 0,Y 664.643,Z 321.429,A -85,B 0,C 180,E1 30240.431,E2 30240.431} C_VEL
LIN {X 0,Y 664.619,Z 321.415,A -85,B 0,C 180,E1 30237.342,E2 30237.342} C_VEL
LIN {X 0,Y 664.647,Z 321.429,A -85,B 0,C 180,E1 30234.302,E2 30234.302} C_VEL
LIN {X 0,Y 664.644,Z 321.443,A -85,B 0,C 180,E1 30231.086,E2 30231.086} C_VEL
LIN {X 0,Y 664.647,Z 321.424,A -85,B 0,C 180,E1 30227.842,E2 30227.842} C_VEL
LIN {X 0,Y 664.682,Z 321.684,A -85,B 0,C 180,E1 30227.71,E2 30227.71} C_VEL
LIN {X 0,Y 666.05,Z 325.108,A -85,B 0,C 180,E1 30227.075,E2 30227.075} C_VEL
LIN {X 0,Y 667.649,Z 327.119,A -85,B 0,C 180,E1 30226.577,E2 30226.577} C_VEL
LIN {X 0,Y 669.346,Z 330.642,A -85,B 0,C 180,E1 30225.907,E2 30225.907} C_VEL
LIN {X 0,Y 670.436,Z 332.063,A -85,B 0,C 180,E1 30225.578,E2 30225.578} C_VEL
LIN {X 0,Y 672.473,Z 336.077,A -85,B 0,C 180,E1 30224.829,E2 30224.829} C_VEL
LIN {X 0,Y 673.644,Z 338.324,A -85,B 0,C 180,E1 30224.415,E2 30224.415} C_VEL
LIN {X 0,Y 676.134,Z 342.748,A -85,B 0,C 180,E1 30223.593,E2 30223.593} C_VEL
LIN {X 0,Y 681.167,Z 352.198,A -85,B 0,C 180,E1 30221.957,E2 30221.957} C_VEL
LIN {X 0,Y 687.996,Z 365.384,A -85,B 0,C 180,E1 30219.852,E2 30219.852} C_VEL
LIN {X 0,Y 689.865,Z 369.149,A -85,B 0,C 180,E1 30219.289,E2 30219.289} C_VEL
LIN {X 0,Y 687.762,Z 402.971,A -85,B 0,C 180,E1 30216.616,E2 30216.616} C_VEL
LIN {X 0,Y 685.601,Z 439.577,A -85,B 0,C 180,E1 30213.868,E2 30213.868} C_VEL
LIN {X 0,Y 683.478,Z 478.366,A -85,B 0,C 180,E1 30211.085,E2 30211.085} C_VEL
LIN {X 0,Y 681.373,Z 519.467,A -85,B 0,C 180,E1 30208.258,E2 30208.258} C_VEL
LIN {X 0,Y 680.313,Z 549.936,A -85,B 0,C 180,E1 30206.199,E2 30206.199} C_VEL
LIN {X 0,Y 681.517,Z 563.206,A -85,B 0,C 180,E1 30205.199,E2 30205.199} C_VEL
LIN {X 0,Y 684.358,Z 574.45,A -85,B 0,C 180,E1 30204.237,E2 30204.237} C_VEL
LIN {X 0,Y 688.458,Z 583.581,A -85,B 0,C 180,E1 30203.35,E2 30203.35} C_VEL
LIN {X 0,Y 694.082,Z 591.605,A -85,B 0,C 180,E1 30202.456,E2 30202.456} C_VEL
LIN {X 0,Y 701.29,Z 598.417,A -85,B 0,C 180,E1 30201.564,E2 30201.564} C_VEL
LIN {X 0,Y 709.471,Z 603.574,A -85,B 0,C 180,E1 30200.743,E2 30200.743} C_VEL
LIN {X 0,Y 714.017,Z 605.501,A -85,B 0,C 180,E1 30200.314,E2 30200.314} C_VEL
LIN {X 0,Y 717.16,Z 606.073,A -85,B 0,C 180,E1 30199.899,E2 30199.899} C_VEL
LIN {X 0,Y 719.477,Z 605.525,A -85,B 0,C 180,E1 30199.428,E2 30199.428} C_VEL
LIN {X 0,Y 720.569,Z 604.038,A -85,B 0,C 180,E1 30198.977,E2 30198.977} C_VEL
LIN {X 0,Y 720.445,Z 601.208,A -85,B 0,C 180,E1 30198.475,E2 30198.475} C_VEL
LIN {X 0,Y 718.806,Z 597.451,A -85,B 0,C 180,E1 30198.029,E2 30198.029} C_VEL
LIN {X 0,Y 715.808,Z 592.991,A -85,B 0,C 180,E1 30197.676,E2 30197.676} C_VEL
LIN {X 0,Y 708.332,Z 582.375,A -85,B 0,C 180,E1 30197.119,E2 30197.119} C_VEL
LIN {X 0,Y 702.038,Z 570.552,A -85,B 0,C 180,E1 30196.64,E2 30196.64} C_VEL
LIN {X 0,Y 696.83,Z 557.31,A -85,B 0,C 180,E1 30196.235,E2 30196.235} C_VEL
LIN {X 0,Y 692.869,Z 542.995,A -85,B 0,C 180,E1 30195.92,E2 30195.92} C_VEL
LIN {X 0,Y 690.135,Z 527.438,A -85,B 0,C 180,E1 30195.7,E2 30195.7} C_VEL
LIN {X 0,Y 688.656,Z 510.427,A -85,B 0,C 180,E1 30195.58,E2 30195.58} C_VEL
LIN {X 0,Y 688.384,Z 487.912,A -85,B 0,C 180,E1 30195.558,E2 30195.558} C_VEL
LIN {X 0,Y 688.52,Z 401.549,A -85,B 0,C 180,E1 30195.545,E2 30195.545} C_VEL
LIN {X 0,Y 689.131,Z 401.217,A -85,B 0,C 180,E1 30195.498,E2 30195.498} C_VEL
LIN {X 0,Y 686.268,Z 610.952,A -85,B 0,C 180,E1 30192.741,E2 30192.741} C_VEL
LIN {X 0,Y 683.413,Z 827.969,A -85,B 0,C 180,E1 30189.955,E2 30189.955} C_VEL
LIN {X 0,Y 682.608,Z 854.74,A -85,B 0,C 180,E1 30189.475,E2 30189.475} C_VEL
LIN {X 0,Y 681.558,Z 881.117,A -85,B 0,C 180,E1 30188.84,E2 30188.84} C_VEL
LIN {X 0,Y 680.359,Z 905.782,A -85,B 0,C 180,E1 30188.084,E2 30188.084} C_VEL
LIN {X 0,Y 678.963,Z 931.454,A -85,B 0,C 180,E1 30187.14,E2 30187.14} C_VEL
LIN {X 0,Y 677.364,Z 957.776,A -85,B 0,C 180,E1 30185.978,E2 30185.978} C_VEL
LIN {X 0,Y 675.903,Z 980.574,A -85,B 0,C 180,E1 30184.811,E2 30184.811} C_VEL
LIN {X 0,Y 674.297,Z 1004.22,A -85,B 0,C 180,E1 30183.426,E2 30183.426} C_VEL
LIN {X 0,Y 672.671,Z 1026.662,A -85,B 0,C 180,E1 30181.922,E2 30181.922} C_VEL
LIN {X 0,Y 671.194,Z 1048.327,A -85,B 0,C 180,E1 30180.281,E2 30180.281} C_VEL
LIN {X 0,Y 669.703,Z 1069.934,A -85,B 0,C 180,E1 30178.43,E2 30178.43} C_VEL
LIN {X 0,Y 668.454,Z 1088.607,A -85,B 0,C 180,E1 30176.628,E2 30176.628} C_VEL
LIN {X 0,Y 667.268,Z 1107.948,A -85,B 0,C 180,E1 30174.523,E2 30174.523} C_VEL
LIN {X 0,Y 666.429,Z 1123.051,A -85,B 0,C 180,E1 30172.671,E2 30172.671} C_VEL
LIN {X 0,Y 665.685,Z 1138.349,A -85,B 0,C 180,E1 30170.576,E2 30170.576} C_VEL
LIN {X 0,Y 665.046,Z 1152.684,A -85,B 0,C 180,E1 30168.313,E2 30168.313} C_VEL
LIN {X 0,Y 664.63,Z 1163.622,A -85,B 0,C 180,E1 30166.338,E2 30166.338} C_VEL
LIN {X 0,Y 664.342,Z 1173.977,A -85,B 0,C 180,E1 30164.2,E2 30164.2} C_VEL
LIN {X 0,Y 664.11,Z 1183.964,A -85,B 0,C 180,E1 30161.726,E2 30161.726} C_VEL
LIN {X 0,Y 664.001,Z 1191.414,A -85,B 0,C 180,E1 30159.446,E2 30159.446} C_VEL
LIN {X 0,Y 663.943,Z 1197.339,A -85,B 0,C 180,E1 30157.092,E2 30157.092} C_VEL
LIN {X 0,Y 663.917,Z 1201.421,A -85,B 0,C 180,E1 30154.837,E2 30154.837} C_VEL
LIN {X 0,Y 663.908,Z 1203.984,A -85,B 0,C 180,E1 30152.589,E2 30152.589} C_VEL
LIN {X 0,Y 663.894,Z 1204.934,A -85,B 0,C 180,E1 30150.344,E2 30150.344} C_VEL
LIN {X 0,Y 663.912,Z 1204.319,A -85,B 0,C 180,E1 30147.928,E2 30147.928} C_VEL
LIN {X 0,Y 663.917,Z 1202.162,A -85,B 0,C 180,E1 30145.68,E2 30145.68} C_VEL
LIN {X 0,Y 663.933,Z 1198.426,A -85,B 0,C 180,E1 30143.427,E2 30143.427} C_VEL
LIN {X 0,Y 663.976,Z 1193.105,A -85,B 0,C 180,E1 30141.163,E2 30141.163} C_VEL
LIN {X 0,Y 664.073,Z 1185.828,A -85,B 0,C 180,E1 30138.799,E2 30138.799} C_VEL
LIN {X 0,Y 664.269,Z 1177.025,A -85,B 0,C 180,E1 30136.506,E2 30136.506} C_VEL
LIN {X 0,Y 664.577,Z 1165.938,A -85,B 0,C 180,E1 30134.107,E2 30134.107} C_VEL
LIN {X 0,Y 664.967,Z 1154.761,A -85,B 0,C 180,E1 30132.045,E2 30132.045} C_VEL
LIN {X 0,Y 665.54,Z 1141.367,A -85,B 0,C 180,E1 30129.876,E2 30129.876} C_VEL
LIN {X 0,Y 666.335,Z 1124.936,A -85,B 0,C 180,E1 30127.572,E2 30127.572} C_VEL
LIN {X 0,Y 667.118,Z 1110.27,A -85,B 0,C 180,E1 30125.752,E2 30125.752} C_VEL
LIN {X 0,Y 668.237,Z 1092.847,A -85,B 0,C 180,E1 30123.805,E2 30123.805} C_VEL
LIN {X 0,Y 669.446,Z 1073.347,A -85,B 0,C 180,E1 30121.885,E2 30121.885} C_VEL
LIN {X 0,Y 670.924,Z 1052.386,A -85,B 0,C 180,E1 30120.049,E2 30120.049} C_VEL
LIN {X 0,Y 672.44,Z 1030.265,A -85,B 0,C 180,E1 30118.338,E2 30118.338} C_VEL
LIN {X 0,Y 673.877,Z 1009.348,A -85,B 0,C 180,E1 30116.904,E2 30116.904} C_VEL
LIN {X 0,Y 675.627,Z 984.752,A -85,B 0,C 180,E1 30115.419,E2 30115.419} C_VEL
LIN {X 0,Y 677.13,Z 961.712,A -85,B 0,C 180,E1 30114.214,E2 30114.214} C_VEL
LIN {X 0,Y 678.51,Z 939.558,A -85,B 0,C 180,E1 30113.198,E2 30113.198} C_VEL
LIN {X 0,Y 679.936,Z 914.175,A -85,B 0,C 180,E1 30112.203,E2 30112.203} C_VEL
LIN {X 0,Y 681.273,Z 887.213,A -85,B 0,C 180,E1 30111.335,E2 30111.335} C_VEL
LIN {X 0,Y 682.391,Z 860.451,A -85,B 0,C 180,E1 30110.65,E2 30110.65} C_VEL
LIN {X 0,Y 683.256,Z 834.086,A -85,B 0,C 180,E1 30110.138,E2 30110.138} C_VEL
LIN {X 0,Y 683.964,Z 793.596,A -85,B 0,C 180,E1 30109.595,E2 30109.595} C_VEL
LIN {X 0,Y 686.853,Z 567.243,A -85,B 0,C 180,E1 30106.692,E2 30106.692} C_VEL
LIN {X 0,Y 689.423,Z 391.341,A -85,B 0,C 180,E1 30104.355,E2 30104.355} C_VEL
LIN {X 0,Y 690.828,Z 388.342,A -85,B 0,C 180,E1 30104.229,E2 30104.229} C_VEL
LIN {X 0,Y 693.608,Z 375.717,A -85,B 0,C 180,E1 30103.98,E2 30103.98} C_VEL
LIN {X 0,Y 696.614,Z 357.881,A -85,B 0,C 180,E1 30103.722,E2 30103.722} C_VEL
LIN {X 0,Y 697.473,Z 357.325,A -85,B 0,C 180,E1 30103.617,E2 30103.617} C_VEL
LIN {X 0,Y 699.856,Z 359.193,A -85,B 0,C 180,E1 30103.167,E2 30103.167} C_VEL
LIN {X 0,Y 700.925,Z 360.297,A -85,B 0,C 180,E1 30102.657,E2 30102.657} C_VEL
LIN {X 0,Y 700.509,Z 360.579,A -85,B 0,C 180,E1 30102.134,E2 30102.134} C_VEL
LIN {X 0,Y 698.579,Z 359.993,A -85,B 0,C 180,E1 30101.616,E2 30101.616} C_VEL
LIN {X 0,Y 695.252,Z 358.441,A -85,B 0,C 180,E1 30101.145,E2 30101.145} C_VEL
LIN {X 0,Y 689.08,Z 354.174,A -85,B 0,C 180,E1 30100.493,E2 30100.493} C_VEL
LIN {X 0,Y 681.487,Z 346.36,A -85,B 0,C 180,E1 30099.606,E2 30099.606} C_VEL
LIN {X 0,Y 674.654,Z 336.726,A -85,B 0,C 180,E1 30098.715,E2 30098.715} C_VEL
LIN {X 0,Y 671.438,Z 332.069,A -85,B 0,C 180,E1 30098.28,E2 30098.28} C_VEL
LIN {X 0,Y 668.77,Z 328.313,A -85,B 0,C 180,E1 30097.915,E2 30097.915} C_VEL
LIN {X 0,Y 667.859,Z 326.888,A -85,B 0,C 180,E1 30097.786,E2 30097.786} C_VEL
LIN {X 0,Y 665.415,Z 323.999,A -85,B 0,C 180,E1 30097.46,E2 30097.46} C_VEL
LIN {X 0,Y 664.621,Z 321.403,A -85,B 0,C 180,E1 30097.293,E2 30097.293} C_VEL
LIN {X 0,Y 664.645,Z 321.444,A -85,B 0,C 180,E1 30094.011,E2 30094.011} C_VEL
LIN {X 0,Y 664.635,Z 321.402,A -85,B 0,C 180,E1 30090.96,E2 30090.96} C_VEL
LIN {X 0,Y 664.632,Z 321.443,A -85,B 0,C 180,E1 30087.797,E2 30087.797} C_VEL
LIN {X 0,Y 664.641,Z 321.401,A -85,B 0,C 180,E1 30084.723,E2 30084.723} C_VEL
LIN {X 0,Y 664.617,Z 321.444,A -85,B 0,C 180,E1 30081.629,E2 30081.629} C_VEL
LIN {X 0,Y 664.618,Z 321.445,A -85,B 0,C 180,E1 30078.69,E2 30078.69} C_VEL
LIN {X 0,Y 664.641,Z 321.443,A -85,B 0,C 180,E1 30075.672,E2 30075.672} C_VEL
LIN {X 0,Y 664.613,Z 321.447,A -85,B 0,C 180,E1 30072.689,E2 30072.689} C_VEL
LIN {X 0,Y 664.615,Z 321.449,A -85,B 0,C 180,E1 30072.302,E2 30072.302} C_VEL
LIN {X 0,Y 666.813,Z 330.501,A -85,B 0,C 180,E1 30071.943,E2 30071.943} C_VEL
LIN {X 0,Y 666.875,Z 403.249,A -85,B 0,C 180,E1 30069.45,E2 30069.45} C_VEL
LIN {X 0,Y 667.26,Z 484.465,A -85,B 0,C 180,E1 30066.539,E2 30066.539} C_VEL
LIN {X 0,Y 667.495,Z 553.242,A -85,B 0,C 180,E1 30063.994,E2 30063.994} C_VEL
LIN {X 0,Y 667.275,Z 634.773,A -85,B 0,C 180,E1 30060.902,E2 30060.902} C_VEL
LIN {X 0,Y 666.766,Z 712.604,A -85,B 0,C 180,E1 30057.894,E2 30057.894} C_VEL
LIN {X 0,Y 666.136,Z 790.851,A -85,B 0,C 180,E1 30054.833,E2 30054.833} C_VEL
LIN {X 0,Y 665.632,Z 842.631,A -85,B 0,C 180,E1 30052.819,E2 30052.819} C_VEL
LIN {X 0,Y 665.295,Z 956.879,A -85,B 0,C 180,E1 30051.557,E2 30051.557} C_VEL
LIN {X 0,Y 665.249,Z 969.317,A -85,B 0,C 180,E1 30051.304,E2 30051.304} C_VEL
LIN {X 0,Y 665.18,Z 980.696,A -85,B 0,C 180,E1 30050.966,E2 30050.966} C_VEL
LIN {X 0,Y 665.081,Z 991.995,A -85,B 0,C 180,E1 30050.52,E2 30050.52} C_VEL
LIN {X 0,Y 664.922,Z 1004.76,A -85,B 0,C 180,E1 30049.867,E2 30049.867} C_VEL
LIN {X 0,Y 664.758,Z 1016.379,A -85,B 0,C 180,E1 30049.075,E2 30049.075} C_VEL
LIN {X 0,Y 664.619,Z 1025.001,A -85,B 0,C 180,E1 30048.351,E2 30048.351} C_VEL
LIN {X 0,Y 664.495,Z 1032.63,A -85,B 0,C 180,E1 30047.574,E2 30047.574} C_VEL
LIN {X 0,Y 664.388,Z 1039.744,A -85,B 0,C 180,E1 30046.687,E2 30046.687} C_VEL
LIN {X 0,Y 664.283,Z 1047.036,A -85,B 0,C 180,E1 30045.53,E2 30045.53} C_VEL
LIN {X 0,Y 664.239,Z 1050.248,A -85,B 0,C 180,E1 30044.861,E2 30044.861} C_VEL
LIN {X 0,Y 663.227,Z 1053.01,A -85,B 0,C 180,E1 30044.241,E2 30044.241} C_VEL
LIN {X 0,Y 659.134,Z 1056.719,A -85,B 0,C 180,E1 30043.18,E2 30043.18} C_VEL
LIN {X 0,Y 656.593,Z 1058.614,A -85,B 0,C 180,E1 30042.348,E2 30042.348} C_VEL
LIN {X 0,Y 656.239,Z 1059.177,A -85,B 0,C 180,E1 30041.964,E2 30041.964} C_VEL
LIN {X 0,Y 656.22,Z 1059.562,A -85,B 0,C 180,E1 30040.692,E2 30040.692} C_VEL
LIN {X 0,Y 656.229,Z 1058.515,A -85,B 0,C 180,E1 30039.566,E2 30039.566} C_VEL
LIN {X 0,Y 656.233,Z 1056.436,A -85,B 0,C 180,E1 30038.55,E2 30038.55} C_VEL
LIN {X 0,Y 656.268,Z 1053.138,A -85,B 0,C 180,E1 30037.516,E2 30037.516} C_VEL
LIN {X 0,Y 656.329,Z 1048.063,A -85,B 0,C 180,E1 30036.38,E2 30036.38} C_VEL
LIN {X 0,Y 656.441,Z 1040.79,A -85,B 0,C 180,E1 30035.207,E2 30035.207} C_VEL
LIN {X 0,Y 656.561,Z 1033.377,A -85,B 0,C 180,E1 30034.276,E2 30034.276} C_VEL
LIN {X 0,Y 656.691,Z 1025.348,A -85,B 0,C 180,E1 30033.456,E2 30033.456} C_VEL
LIN {X 0,Y 656.863,Z 1015.454,A -85,B 0,C 180,E1 30032.631,E2 30032.631} C_VEL
LIN {X 0,Y 657.057,Z 1002.58,A -85,B 0,C 180,E1 30031.798,E2 30031.798} C_VEL
LIN {X 0,Y 657.204,Z 991.312,A -85,B 0,C 180,E1 30031.234,E2 30031.234} C_VEL
LIN {X 0,Y 657.307,Z 980.253,A -85,B 0,C 180,E1 30030.801,E2 30030.801} C_VEL
LIN {X 0,Y 657.394,Z 968.337,A -85,B 0,C 180,E1 30030.452,E2 30030.452} C_VEL
LIN {X 0,Y 657.456,Z 953.404,A -85,B 0,C 180,E1 30030.166,E2 30030.166} C_VEL
LIN {X 0,Y 657.844,Z 840.84,A -85,B 0,C 180,E1 30028.909,E2 30028.909} C_VEL
LIN {X 0,Y 658.647,Z 759.885,A -85,B 0,C 180,E1 30025.675,E2 30025.675} C_VEL
LIN {X 0,Y 659.485,Z 680.365,A -85,B 0,C 180,E1 30022.501,E2 30022.501} C_VEL
LIN {X 0,Y 660.226,Z 603.932,A -85,B 0,C 180,E1 30019.452,E2 30019.452} C_VEL
LIN {X 0,Y 660.947,Z 526.398,A -85,B 0,C 180,E1 30016.347,E2 30016.347} C_VEL
LIN {X 0,Y 661.072,Z 512.546,A -85,B 0,C 180,E1 30015.783,E2 30015.783} C_VEL
LIN {X 0,Y 662.249,Z 514.528,A -85,B 0,C 180,E1 30015.648,E2 30015.648} C_VEL
LIN {X 0,Y 663.987,Z 514.657,A -85,B 0,C 180,E1 30015.493,E2 30015.493} C_VEL
LIN {X 0,Y 666.627,Z 512.537,A -85,B 0,C 180,E1 30015.294,E2 30015.294} C_VEL
LIN {X 0,Y 670.188,Z 507.032,A -85,B 0,C 180,E1 30015.069,E2 30015.069} C_VEL
LIN {X 0,Y 670.713,Z 506.069,A -85,B 0,C 180,E1 30015.038,E2 30015.038} C_VEL
LIN {X 0,Y 674.178,Z 504.877,A -85,B 0,C 180,E1 30014.761,E2 30014.761} C_VEL
LIN {X 0,Y 677.934,Z 501.515,A -85,B 0,C 180,E1 30014.495,E2 30014.495} C_VEL
LIN {X 0,Y 681.573,Z 496.665,A -85,B 0,C 180,E1 30014.265,E2 30014.265} C_VEL
LIN {X 0,Y 678.693,Z 702.208,A -85,B 0,C 180,E1 30011.585,E2 30011.585} C_VEL
LIN {X 0,Y 677.231,Z 799.147,A -85,B 0,C 180,E1 30010.327,E2 30010.327} C_VEL
LIN {X 0,Y 676.349,Z 826.448,A -85,B 0,C 180,E1 30009.83,E2 30009.83} C_VEL
LIN {X 0,Y 675.117,Z 853.56,A -85,B 0,C 180,E1 30009.154,E2 30009.154} C_VEL
LIN {X 0,Y 673.944,Z 875.8,A -85,B 0,C 180,E1 30008.464,E2 30008.464} C_VEL
LIN {X 0,Y 672.756,Z 896.56,A -85,B 0,C 180,E1 30007.706,E2 30007.706} C_VEL
LIN {X 0,Y 671.501,Z 916.311,A -85,B 0,C 180,E1 30006.876,E2 30006.876} C_VEL
LIN {X 0,Y 669.966,Z 938.641,A -85,B 0,C 180,E1 30005.806,E2 30005.806} C_VEL
LIN {X 0,Y 668.08,Z 963.985,A -85,B 0,C 180,E1 30004.402,E2 30004.402} C_VEL
LIN {X 0,Y 666.415,Z 986.087,A -85,B 0,C 180,E1 30002.994,E2 30002.994} C_VEL
LIN {X 0,Y 664.707,Z 1008.67,A -85,B 0,C 180,E1 30001.365,E2 30001.365} C_VEL
LIN {X 0,Y 662.915,Z 1031.932,A -85,B 0,C 180,E1 29999.454,E2 29999.454} C_VEL
LIN {X 0,Y 661.41,Z 1052.552,A -85,B 0,C 180,E1 29997.521,E2 29997.521} C_VEL
LIN {X 0,Y 660.145,Z 1070.158,A -85,B 0,C 180,E1 29995.671,E2 29995.671} C_VEL
LIN {X 0,Y 659.002,Z 1088.326,A -85,B 0,C 180,E1 29993.519,E2 29993.519} C_VEL
LIN {X 0,Y 658.159,Z 1102.837,A -85,B 0,C 180,E1 29991.572,E2 29991.572} C_VEL
LIN {X 0,Y 657.543,Z 1114.537,A -85,B 0,C 180,E1 29989.823,E2 29989.823} C_VEL
LIN {X 0,Y 657.069,Z 1124.99,A -85,B 0,C 180,E1 29988.086,E2 29988.086} C_VEL
LIN {X 0,Y 656.678,Z 1134.752,A -85,B 0,C 180,E1 29986.271,E2 29986.271} C_VEL
LIN {X 0,Y 656.353,Z 1144.941,A -85,B 0,C 180,E1 29984.109,E2 29984.109} C_VEL
LIN {X 0,Y 656.125,Z 1154.747,A -85,B 0,C 180,E1 29981.606,E2 29981.606} C_VEL
LIN {X 0,Y 656.007,Z 1161.734,A -85,B 0,C 180,E1 29979.387,E2 29979.387} C_VEL
LIN {X 0,Y 655.948,Z 1167.216,A -85,B 0,C 180,E1 29977.182,E2 29977.182} C_VEL
LIN {X 0,Y 655.92,Z 1171.372,A -85,B 0,C 180,E1 29974.898,E2 29974.898} C_VEL
LIN {X 0,Y 655.907,Z 1174.059,A -85,B 0,C 180,E1 29972.447,E2 29972.447} C_VEL
LIN {X 0,Y 655.902,Z 1174.957,A -85,B 0,C 180,E1 29970.176,E2 29970.176} C_VEL
LIN {X 0,Y 655.912,Z 1174.231,A -85,B 0,C 180,E1 29967.73,E2 29967.73} C_VEL
LIN {X 0,Y 655.912,Z 1172.003,A -85,B 0,C 180,E1 29965.455,E2 29965.455} C_VEL
LIN {X 0,Y 655.936,Z 1167.811,A -85,B 0,C 180,E1 29962.997,E2 29962.997} C_VEL
LIN {X 0,Y 655.992,Z 1162.484,A -85,B 0,C 180,E1 29960.792,E2 29960.792} C_VEL
LIN {X 0,Y 656.095,Z 1155.958,A -85,B 0,C 180,E1 29958.663,E2 29958.663} C_VEL
LIN {X 0,Y 656.263,Z 1148.264,A -85,B 0,C 180,E1 29956.611,E2 29956.611} C_VEL
LIN {X 0,Y 656.558,Z 1138.401,A -85,B 0,C 180,E1 29954.363,E2 29954.363} C_VEL
LIN {X 0,Y 657.004,Z 1126.557,A -85,B 0,C 180,E1 29952.097,E2 29952.097} C_VEL
LIN {X 0,Y 657.488,Z 1115.7,A -85,B 0,C 180,E1 29950.27,E2 29950.27} C_VEL
LIN {X 0,Y 658.083,Z 1104.119,A -85,B 0,C 180,E1 29948.522,E2 29948.522} C_VEL
LIN {X 0,Y 658.811,Z 1091.179,A -85,B 0,C 180,E1 29946.76,E2 29946.76} C_VEL
LIN {X 0,Y 659.913,Z 1074.35,A -85,B 0,C 180,E1 29944.706,E2 29944.706} C_VEL
LIN {X 0,Y 661.219,Z 1055.004,A -85,B 0,C 180,E1 29942.634,E2 29942.634} C_VEL
LIN {X 0,Y 662.611,Z 1036.095,A -85,B 0,C 180,E1 29940.831,E2 29940.831} C_VEL
LIN {X 0,Y 664.155,Z 1015.447,A -85,B 0,C 180,E1 29939.076,E2 29939.076} C_VEL
LIN {X 0,Y 665.97,Z 992.187,A -85,B 0,C 180,E1 29937.335,E2 29937.335} C_VEL
LIN {X 0,Y 667.696,Z 969.367,A -85,B 0,C 180,E1 29935.837,E2 29935.837} C_VEL
LIN {X 0,Y 669.292,Z 947.604,A -85,B 0,C 180,E1 29934.576,E2 29934.576} C_VEL
LIN {X 0,Y 671.184,Z 921.092,A -85,B 0,C 180,E1 29933.246,E2 29933.246} C_VEL
LIN {X 0,Y 672.665,Z 897.996,A -85,B 0,C 180,E1 29932.26,E2 29932.26} C_VEL
LIN {X 0,Y 673.886,Z 876.816,A -85,B 0,C 180,E1 29931.48,E2 29931.48} C_VEL
LIN {X 0,Y 675.073,Z 854.522,A -85,B 0,C 180,E1 29930.784,E2 29930.784} C_VEL
LIN {X 0,Y 676.255,Z 828.632,A -85,B 0,C 180,E1 29930.129,E2 29930.129} C_VEL
LIN {X 0,Y 677.204,Z 800.345,A -85,B 0,C 180,E1 29929.601,E2 29929.601} C_VEL
LIN {X 0,Y 678.308,Z 730.544,A -85,B 0,C 180,E1 29928.688,E2 29928.688} C_VEL
LIN {X 0,Y 681.41,Z 509.816,A -85,B 0,C 180,E1 29925.821,E2 29925.821} C_VEL
LIN {X 0,Y 683.599,Z 361.261,A -85,B 0,C 180,E1 29923.835,E2 29923.835} C_VEL
LIN {X 0,Y 671.35,Z 343.31,A -85,B 0,C 180,E1 29922.459,E2 29922.459} C_VEL
LIN {X 0,Y 666.715,Z 337.216,A -85,B 0,C 180,E1 29921.923,E2 29921.923} C_VEL
LIN {X 0,Y 662.193,Z 332.424,A -85,B 0,C 180,E1 29921.404,E2 29921.404} C_VEL
LIN {X 0,Y 661.288,Z 331.538,A -85,B 0,C 180,E1 29921.243,E2 29921.243} C_VEL
LIN {X 0,Y 659.702,Z 328.279,A -85,B 0,C 180,E1 29920.559,E2 29920.559} C_VEL
LIN {X 0,Y 658.863,Z 326.969,A -85,B 0,C 180,E1 29920.242,E2 29920.242} C_VEL
LIN {X 0,Y 657.032,Z 323.87,A -85,B 0,C 180,E1 29919.504,E2 29919.504} C_VEL
LIN {X 0,Y 656.709,Z 322.432,A -85,B 0,C 180,E1 29919.199,E2 29919.199} C_VEL
LIN {X 0,Y 656.679,Z 322.428,A -85,B 0,C 180,E1 29916.199,E2 29916.199} C_VEL
LIN {X 0,Y 656.693,Z 322.4,A -85,B 0,C 180,E1 29913.133,E2 29913.133} C_VEL
LIN {X 0,Y 656.683,Z 322.41,A -85,B 0,C 180,E1 29910.137,E2 29910.137} C_VEL
LIN {X 0,Y 656.708,Z 322.433,A -85,B 0,C 180,E1 29907.179,E2 29907.179} C_VEL
LIN {X 0,Y 656.702,Z 322.407,A -85,B 0,C 180,E1 29903.987,E2 29903.987} C_VEL
LIN {X 0,Y 656.704,Z 322.404,A -85,B 0,C 180,E1 29900.798,E2 29900.798} C_VEL
LIN {X 0,Y 656.689,Z 322.434,A -85,B 0,C 180,E1 29897.73,E2 29897.73} C_VEL
LIN {X 0,Y 656.708,Z 322.41,A -85,B 0,C 180,E1 29894.55,E2 29894.55} C_VEL
LIN {X 0,Y 656.677,Z 322.409,A -85,B 0,C 180,E1 29891.595,E2 29891.595} C_VEL
LIN {X 0,Y 656.699,Z 322.434,A -85,B 0,C 180,E1 29888.581,E2 29888.581} C_VEL
LIN {X 0,Y 656.683,Z 322.406,A -85,B 0,C 180,E1 29885.505,E2 29885.505} C_VEL
LIN {X 0,Y 656.702,Z 322.408,A -85,B 0,C 180,E1 29882.443,E2 29882.443} C_VEL
LIN {X 0,Y 656.71,Z 322.432,A -85,B 0,C 180,E1 29879.302,E2 29879.302} C_VEL
LIN {X 0,Y 656.707,Z 322.416,A -85,B 0,C 180,E1 29875.984,E2 29875.984} C_VEL
LIN {X 0,Y 656.676,Z 322.399,A -85,B 0,C 180,E1 29873.003,E2 29873.003} C_VEL
LIN {X 0,Y 656.701,Z 322.402,A -85,B 0,C 180,E1 29869.916,E2 29869.916} C_VEL
LIN {X 0,Y 656.718,Z 322.622,A -85,B 0,C 180,E1 29869.029,E2 29869.029} C_VEL
LIN {X 0,Y 658.132,Z 326.058,A -85,B 0,C 180,E1 29868.342,E2 29868.342} C_VEL
LIN {X 0,Y 659.706,Z 327.903,A -85,B 0,C 180,E1 29867.838,E2 29867.838} C_VEL
LIN {X 0,Y 661.232,Z 331.423,A -85,B 0,C 180,E1 29867.156,E2 29867.156} C_VEL
LIN {X 0,Y 662.745,Z 333.562,A -85,B 0,C 180,E1 29866.654,E2 29866.654} C_VEL
LIN {X 0,Y 664.787,Z 337.3,A -85,B 0,C 180,E1 29865.897,E2 29865.897} C_VEL
LIN {X 0,Y 668.525,Z 344.236,A -85,B 0,C 180,E1 29864.56,E2 29864.56} C_VEL
LIN {X 0,Y 673.48,Z 353.278,A -85,B 0,C 180,E1 29862.905,E2 29862.905} C_VEL
LIN {X 0,Y 680.643,Z 367.122,A -85,B 0,C 180,E1 29860.61,E2 29860.61} C_VEL
LIN {X 0,Y 684.085,Z 374.185,A -85,B 0,C 180,E1 29859.534,E2 29859.534} C_VEL
LIN {X 0,Y 681.845,Z 407.253,A -85,B 0,C 180,E1 29856.904,E2 29856.904} C_VEL
LIN {X 0,Y 679.482,Z 443.932,A -85,B 0,C 180,E1 29854.131,E2 29854.131} C_VEL
LIN {X 0,Y 677.136,Z 483.208,A -85,B 0,C 180,E1 29851.294,E2 29851.294} C_VEL
LIN {X 0,Y 674.829,Z 524.649,A -85,B 0,C 180,E1 29848.424,E2 29848.424} C_VEL
LIN {X 0,Y 673.76,Z 552.967,A -85,B 0,C 180,E1 29846.491,E2 29846.491} C_VEL
LIN {X 0,Y 674.964,Z 566.871,A -85,B 0,C 180,E1 29845.432,E2 29845.432} C_VEL
LIN {X 0,Y 677.724,Z 578.184,A -85,B 0,C 180,E1 29844.458,E2 29844.458} C_VEL
LIN {X 0,Y 681.698,Z 587.482,A -85,B 0,C 180,E1 29843.556,E2 29843.556} C_VEL
LIN {X 0,Y 687.657,Z 596.377,A -85,B 0,C 180,E1 29842.57,E2 29842.57} C_VEL
LIN {X 0,Y 695.327,Z 603.869,A -85,B 0,C 180,E1 29841.594,E2 29841.594} C_VEL
LIN {X 0,Y 704.072,Z 609.559,A -85,B 0,C 180,E1 29840.699,E2 29840.699} C_VEL
LIN {X 0,Y 710.69,Z 612.385,A -85,B 0,C 180,E1 29840.092,E2 29840.092} C_VEL
LIN {X 0,Y 713.884,Z 612.892,A -85,B 0,C 180,E1 29839.677,E2 29839.677} C_VEL
LIN {X 0,Y 716.238,Z 612.315,A -85,B 0,C 180,E1 29839.206,E2 29839.206} C_VEL
LIN {X 0,Y 717.426,Z 610.54,A -85,B 0,C 180,E1 29838.693,E2 29838.693} C_VEL
LIN {X 0,Y 717.147,Z 607.6,A -85,B 0,C 180,E1 29838.194,E2 29838.194} C_VEL
LIN {X 0,Y 715.34,Z 603.775,A -85,B 0,C 180,E1 29837.752,E2 29837.752} C_VEL
LIN {X 0,Y 712.186,Z 599.314,A -85,B 0,C 180,E1 29837.407,E2 29837.407} C_VEL
LIN {X 0,Y 704.495,Z 588.556,A -85,B 0,C 180,E1 29836.829,E2 29836.829} C_VEL
LIN {X 0,Y 697.869,Z 576.398,A -85,B 0,C 180,E1 29836.316,E2 29836.316} C_VEL
LIN {X 0,Y 692.33,Z 562.795,A -85,B 0,C 180,E1 29835.877,E2 29835.877} C_VEL
LIN {X 0,Y 688.018,Z 548.029,A -85,B 0,C 180,E1 29835.528,E2 29835.528} C_VEL
LIN {X 0,Y 684.989,Z 532.232,A -85,B 0,C 180,E1 29835.278,E2 29835.278} C_VEL
LIN {X 0,Y 683.204,Z 515.044,A -85,B 0,C 180,E1 29835.13,E2 29835.13} C_VEL
LIN {X 0,Y 682.697,Z 495.882,A -85,B 0,C 180,E1 29835.088,E2 29835.088} C_VEL
LIN {X 0,Y 682.661,Z 469.27,A -85,B 0,C 180,E1 29835.085,E2 29835.085} C_VEL
LIN {X 0,Y 682.453,Z 470.233,A -85,B 0,C 180,E1 29835.056,E2 29835.056} C_VEL
LIN {X 0,Y 679.355,Z 684.371,A -85,B 0,C 180,E1 29832.246,E2 29832.246} C_VEL
LIN {X 0,Y 677.238,Z 829.238,A -85,B 0,C 180,E1 29830.372,E2 29830.372} C_VEL
LIN {X 0,Y 676.328,Z 856.37,A -85,B 0,C 180,E1 29829.874,E2 29829.874} C_VEL
LIN {X 0,Y 675.182,Z 882.879,A -85,B 0,C 180,E1 29829.222,E2 29829.222} C_VEL
LIN {X 0,Y 673.857,Z 907.917,A -85,B 0,C 180,E1 29828.44,E2 29828.44} C_VEL
LIN {X 0,Y 672.254,Z 934.518,A -85,B 0,C 180,E1 29827.437,E2 29827.437} C_VEL
LIN {X 0,Y 670.632,Z 958.777,A -85,B 0,C 180,E1 29826.344,E2 29826.344} C_VEL
LIN {X 0,Y 669.002,Z 982.212,A -85,B 0,C 180,E1 29825.127,E2 29825.127} C_VEL
LIN {X 0,Y 667.179,Z 1006.473,A -85,B 0,C 180,E1 29823.675,E2 29823.675} C_VEL
LIN {X 0,Y 665.408,Z 1028.979,A -85,B 0,C 180,E1 29822.135,E2 29822.135} C_VEL
LIN {X 0,Y 663.785,Z 1050.658,A -85,B 0,C 180,E1 29820.455,E2 29820.455} C_VEL
LIN {X 0,Y 662.178,Z 1071.852,A -85,B 0,C 180,E1 29818.597,E2 29818.597} C_VEL
LIN {X 0,Y 660.84,Z 1090.256,A -85,B 0,C 180,E1 29816.784,E2 29816.784} C_VEL
LIN {X 0,Y 659.593,Z 1108.729,A -85,B 0,C 180,E1 29814.732,E2 29814.732} C_VEL
LIN {X 0,Y 658.708,Z 1122.991,A -85,B 0,C 180,E1 29812.96,E2 29812.96} C_VEL
LIN {X 0,Y 657.877,Z 1138.453,A -85,B 0,C 180,E1 29810.816,E2 29810.816} C_VEL
LIN {X 0,Y 657.179,Z 1152.687,A -85,B 0,C 180,E1 29808.54,E2 29808.54} C_VEL
LIN {X 0,Y 656.717,Z 1163.624,A -85,B 0,C 180,E1 29806.541,E2 29806.541} C_VEL
LIN {X 0,Y 656.394,Z 1174.128,A -85,B 0,C 180,E1 29804.343,E2 29804.343} C_VEL
LIN {X 0,Y 656.129,Z 1183.965,A -85,B 0,C 180,E1 29801.871,E2 29801.871} C_VEL
LIN {X 0,Y 656.01,Z 1191.468,A -85,B 0,C 180,E1 29799.543,E2 29799.543} C_VEL
LIN {X 0,Y 655.949,Z 1197.338,A -85,B 0,C 180,E1 29797.179,E2 29797.179} C_VEL
LIN {X 0,Y 655.92,Z 1201.42,A -85,B 0,C 180,E1 29794.896,E2 29794.896} C_VEL
LIN {X 0,Y 655.909,Z 1203.983,A -85,B 0,C 180,E1 29792.62,E2 29792.62} C_VEL
LIN {X 0,Y 655.894,Z 1204.934,A -85,B 0,C 180,E1 29790.348,E2 29790.348} C_VEL
LIN {X 0,Y 655.913,Z 1204.319,A -85,B 0,C 180,E1 29787.902,E2 29787.902} C_VEL
LIN {X 0,Y 655.916,Z 1202.161,A -85,B 0,C 180,E1 29785.628,E2 29785.628} C_VEL
LIN {X 0,Y 655.933,Z 1198.427,A -85,B 0,C 180,E1 29783.346,E2 29783.346} C_VEL
LIN {X 0,Y 655.984,Z 1193.103,A -85,B 0,C 180,E1 29781.055,E2 29781.055} C_VEL
LIN {X 0,Y 656.1,Z 1185.826,A -85,B 0,C 180,E1 29778.661,E2 29778.661} C_VEL
LIN {X 0,Y 656.31,Z 1177.03,A -85,B 0,C 180,E1 29776.34,E2 29776.34} C_VEL
LIN {X 0,Y 656.65,Z 1165.94,A -85,B 0,C 180,E1 29773.91,E2 29773.91} C_VEL
LIN {X 0,Y 657.089,Z 1154.764,A -85,B 0,C 180,E1 29771.823,E2 29771.823} C_VEL
LIN {X 0,Y 657.732,Z 1141.365,A -85,B 0,C 180,E1 29769.626,E2 29769.626} C_VEL
LIN {X 0,Y 658.603,Z 1125.106,A -85,B 0,C 180,E1 29767.317,E2 29767.317} C_VEL
LIN {X 0,Y 659.481,Z 1110.27,A -85,B 0,C 180,E1 29765.453,E2 29765.453} C_VEL
LIN {X 0,Y 660.7,Z 1092.845,A -85,B 0,C 180,E1 29763.483,E2 29763.483} C_VEL
LIN {X 0,Y 662.075,Z 1073.082,A -85,B 0,C 180,E1 29761.518,E2 29761.518} C_VEL
LIN {X 0,Y 663.697,Z 1051.924,A -85,B 0,C 180,E1 29759.649,E2 29759.649} C_VEL
LIN {X 0,Y 665.317,Z 1030.212,A -85,B 0,C 180,E1 29757.955,E2 29757.955} C_VEL
LIN {X 0,Y 666.918,Z 1009.35,A -85,B 0,C 180,E1 29756.513,E2 29756.513} C_VEL
LIN {X 0,Y 668.748,Z 985.596,A -85,B 0,C 180,E1 29755.064,E2 29755.064} C_VEL
LIN {X 0,Y 670.446,Z 961.717,A -85,B 0,C 180,E1 29753.801,E2 29753.801} C_VEL
LIN {X 0,Y 672.013,Z 938.45,A -85,B 0,C 180,E1 29752.729,E2 29752.729} C_VEL
LIN {X 0,Y 673.674,Z 911.572,A -85,B 0,C 180,E1 29751.683,E2 29751.683} C_VEL
LIN {X 0,Y 675.061,Z 885.199,A -85,B 0,C 180,E1 29750.846,E2 29750.846} C_VEL
LIN {X 0,Y 676.215,Z 859.041,A -85,B 0,C 180,E1 29750.185,E2 29750.185} C_VEL
LIN {X 0,Y 677.15,Z 832.498,A -85,B 0,C 180,E1 29749.678,E2 29749.678} C_VEL
LIN {X 0,Y 677.993,Z 783.741,A -85,B 0,C 180,E1 29749.029,E2 29749.029} C_VEL
LIN {X 0,Y 681.114,Z 561.009,A -85,B 0,C 180,E1 29746.146,E2 29746.146} C_VEL
LIN {X 0,Y 682.709,Z 462.976,A -85,B 0,C 180,E1 29744.835,E2 29744.835} C_VEL
LIN {X 0,Y 684.829,Z 454.336,A -85,B 0,C 180,E1 29744.601,E2 29744.601} C_VEL
LIN {X 0,Y 688.488,Z 432.492,A -85,B 0,C 180,E1 29744.242,E2 29744.242} C_VEL
LIN {X 0,Y 692.821,Z 400.526,A -85,B 0,C 180,E1 29743.894,E2 29743.894} C_VEL
LIN {X 0,Y 693.587,Z 394.89,A -85,B 0,C 180,E1 29743.833,E2 29743.833} C_VEL
LIN {X 0,Y 695.356,Z 387.752,A -85,B 0,C 180,E1 29743.605,E2 29743.605} C_VEL
LIN {X 0,Y 698.377,Z 369.637,A -85,B 0,C 180,E1 29743.289,E2 29743.289} C_VEL
LIN {X 0,Y 698.768,Z 367.072,A -85,B 0,C 180,E1 29743.252,E2 29743.252} C_VEL
LIN {X 0,Y 699.834,Z 368.161,A -85,B 0,C 180,E1 29742.739,E2 29742.739} C_VEL
LIN {X 0,Y 699.401,Z 368.496,A -85,B 0,C 180,E1 29742.216,E2 29742.216} C_VEL
LIN {X 0,Y 697.449,Z 368.011,A -85,B 0,C 180,E1 29741.699,E2 29741.699} C_VEL
LIN {X 0,Y 694.085,Z 366.661,A -85,B 0,C 180,E1 29741.229,E2 29741.229} C_VEL
LIN {X 0,Y 687.209,Z 362.494,A -85,B 0,C 180,E1 29740.516,E2 29740.516} C_VEL
LIN {X 0,Y 677.974,Z 353.377,A -85,B 0,C 180,E1 29739.441,E2 29739.441} C_VEL
LIN {X 0,Y 667.011,Z 337.964,A -85,B 0,C 180,E1 29737.979,E2 29737.979} C_VEL
LIN {X 0,Y 663.577,Z 333.081,A -85,B 0,C 180,E1 29737.5,E2 29737.5} C_VEL
LIN {X 0,Y 660.891,Z 329.3,A -85,B 0,C 180,E1 29737.119,E2 29737.119} C_VEL
LIN {X 0,Y 660.207,Z 328.075,A -85,B 0,C 180,E1 29737.015,E2 29737.015} C_VEL
LIN {X 0,Y 657.704,Z 325.397,A -85,B 0,C 180,E1 29736.675,E2 29736.675} C_VEL
LIN {X 0,Y 656.703,Z 322.379,A -85,B 0,C 180,E1 29736.463,E2 29736.463} C_VEL
LIN {X 0,Y 656.682,Z 322.432,A -85,B 0,C 180,E1 29733.445,E2 29733.445} C_VEL
LIN {X 0,Y 656.712,Z 322.399,A -85,B 0,C 180,E1 29730.263,E2 29730.263} C_VEL
LIN {X 0,Y 656.697,Z 322.416,A -85,B 0,C 180,E1 29727.18,E2 29727.18} C_VEL
LIN {X 0,Y 656.705,Z 322.411,A -85,B 0,C 180,E1 29723.892,E2 29723.892} C_VEL
LIN {X 0,Y 656.705,Z 322.42,A -85,B 0,C 180,E1 29720.779,E2 29720.779} C_VEL
LIN {X 0,Y 656.693,Z 322.424,A -85,B 0,C 180,E1 29717.546,E2 29717.546} C_VEL
LIN {X 0,Y 656.712,Z 322.432,A -85,B 0,C 180,E1 29714.452,E2 29714.452} C_VEL
LIN {X 0,Y 656.694,Z 322.599,A -85,B 0,C 180,E1 29712.47,E2 29712.47} C_VEL
LIN {X 0,Y 659.112,Z 331.597,A -85,B 0,C 180,E1 29712.107,E2 29712.107} C_VEL
LIN {X 0,Y 659.173,Z 408.355,A -85,B 0,C 180,E1 29709.473,E2 29709.473} C_VEL
LIN {X 0,Y 659.625,Z 493.94,A -85,B 0,C 180,E1 29706.395,E2 29706.395} C_VEL
LIN {X 0,Y 659.77,Z 567.68,A -85,B 0,C 180,E1 29703.649,E2 29703.649} C_VEL
LIN {X 0,Y 659.427,Z 642.28,A -85,B 0,C 180,E1 29700.782,E2 29700.782} C_VEL
LIN {X 0,Y 659.021,Z 712.47,A -85,B 0,C 180,E1 29698.087,E2 29698.087} C_VEL
LIN {X 0,Y 658.365,Z 790.195,A -85,B 0,C 180,E1 29695.034,E2 29695.034} C_VEL
LIN {X 0,Y 657.79,Z 843.502,A -85,B 0,C 180,E1 29692.947,E2 29692.947} C_VEL
LIN {X 0,Y 657.421,Z 958.053,A -85,B 0,C 180,E1 29691.665,E2 29691.665} C_VEL
LIN {X 0,Y 657.384,Z 970.457,A -85,B 0,C 180,E1 29691.409,E2 29691.409} C_VEL
LIN {X 0,Y 657.321,Z 981.682,A -85,B 0,C 180,E1 29691.074,E2 29691.074} C_VEL
LIN {X 0,Y 657.226,Z 992.839,A -85,B 0,C 180,E1 29690.631,E2 29690.631} C_VEL
LIN {X 0,Y 657.076,Z 1005.005,A -85,B 0,C 180,E1 29690.01,E2 29690.01} C_VEL
LIN {X 0,Y 656.904,Z 1016.876,A -85,B 0,C 180,E1 29689.209,E2 29689.209} C_VEL
LIN {X 0,Y 656.759,Z 1025.413,A -85,B 0,C 180,E1 29688.496,E2 29688.496} C_VEL
LIN {X 0,Y 656.62,Z 1033.337,A -85,B 0,C 180,E1 29687.691,E2 29687.691} C_VEL
LIN {X 0,Y 656.51,Z 1039.874,A -85,B 0,C 180,E1 29686.883,E2 29686.883} C_VEL
LIN {X 0,Y 656.41,Z 1045.802,A -85,B 0,C 180,E1 29685.983,E2 29685.983} C_VEL
LIN {X 0,Y 656.332,Z 1051.383,A -85,B 0,C 180,E1 29684.9,E2 29684.9} C_VEL
LIN {X 0,Y 656.267,Z 1055.951,A -85,B 0,C 180,E1 29683.628,E2 29683.628} C_VEL
LIN {X 0,Y 656.238,Z 1058.367,A -85,B 0,C 180,E1 29682.52,E2 29682.52} C_VEL
LIN {X 0,Y 656.239,Z 1059.177,A -85,B 0,C 180,E1 29681.964,E2 29681.964} C_VEL
LIN {X 0,Y 655.243,Z 1059.908,A -85,B 0,C 180,E1 29681.292,E2 29681.292} C_VEL
LIN {X 0,Y 651.348,Z 1060.272,A -85,B 0,C 180,E1 29680.214,E2 29680.214} C_VEL
LIN {X 0,Y 648.737,Z 1059.449,A -85,B 0,C 180,E1 29679.36,E2 29679.36} C_VEL
LIN {X 0,Y 648.312,Z 1058.551,A -85,B 0,C 180,E1 29678.927,E2 29678.927} C_VEL
LIN {X 0,Y 648.348,Z 1055.029,A -85,B 0,C 180,E1 29677.704,E2 29677.704} C_VEL
LIN {X 0,Y 648.391,Z 1051.113,A -85,B 0,C 180,E1 29676.748,E2 29676.748} C_VEL
LIN {X 0,Y 648.463,Z 1045.971,A -85,B 0,C 180,E1 29675.785,E2 29675.785} C_VEL
LIN {X 0,Y 648.572,Z 1039.426,A -85,B 0,C 180,E1 29674.817,E2 29674.817} C_VEL
LIN {X 0,Y 648.753,Z 1030.278,A -85,B 0,C 180,E1 29673.747,E2 29673.747} C_VEL
LIN {X 0,Y 648.929,Z 1020.138,A -85,B 0,C 180,E1 29672.833,E2 29672.833} C_VEL
LIN {X 0,Y 649.07,Z 1010.526,A -85,B 0,C 180,E1 29672.13,E2 29672.13} C_VEL
LIN {X 0,Y 649.235,Z 1000.494,A -85,B 0,C 180,E1 29671.532,E2 29671.532} C_VEL
LIN {X 0,Y 649.381,Z 989.026,A -85,B 0,C 180,E1 29670.986,E2 29670.986} C_VEL
LIN {X 0,Y 649.501,Z 973.526,A -85,B 0,C 180,E1 29670.45,E2 29670.45} C_VEL
LIN {X 0,Y 649.554,Z 960.893,A -85,B 0,C 180,E1 29670.162,E2 29670.162} C_VEL
LIN {X 0,Y 649.583,Z 944.34,A -85,B 0,C 180,E1 29669.937,E2 29669.937} C_VEL
LIN {X 0,Y 650.02,Z 841.806,A -85,B 0,C 180,E1 29668.776,E2 29668.776} C_VEL
LIN {X 0,Y 650.862,Z 763.136,A -85,B 0,C 180,E1 29665.618,E2 29665.618} C_VEL
LIN {X 0,Y 651.745,Z 685.013,A -85,B 0,C 180,E1 29662.478,E2 29662.478} C_VEL
LIN {X 0,Y 652.564,Z 606.471,A -85,B 0,C 180,E1 29659.329,E2 29659.329} C_VEL
LIN {X 0,Y 653.207,Z 535.472,A -85,B 0,C 180,E1 29656.484,E2 29656.484} C_VEL
LIN {X 0,Y 653.337,Z 528.959,A -85,B 0,C 180,E1 29656.208,E2 29656.208} C_VEL
LIN {X 0,Y 654.445,Z 531.044,A -85,B 0,C 180,E1 29656.081,E2 29656.081} C_VEL
LIN {X 0,Y 656.222,Z 531.422,A -85,B 0,C 180,E1 29655.927,E2 29655.927} C_VEL
LIN {X 0,Y 658.859,Z 529.29,A -85,B 0,C 180,E1 29655.725,E2 29655.725} C_VEL
LIN {X 0,Y 662.453,Z 523.676,A -85,B 0,C 180,E1 29655.492,E2 29655.492} C_VEL
LIN {X 0,Y 662.93,Z 522.723,A -85,B 0,C 180,E1 29655.464,E2 29655.464} C_VEL
LIN {X 0,Y 666.371,Z 521.536,A -85,B 0,C 180,E1 29655.181,E2 29655.181} C_VEL
LIN {X 0,Y 670.103,Z 518.189,A -85,B 0,C 180,E1 29654.91,E2 29654.91} C_VEL
LIN {X 0,Y 673.633,Z 513.242,A -85,B 0,C 180,E1 29654.684,E2 29654.684} C_VEL
LIN {X 0,Y 675.635,Z 512.447,A -85,B 0,C 180,E1 29654.528,E2 29654.528} C_VEL
LIN {X 0,Y 672.147,Z 740.714,A -85,B 0,C 180,E1 29651.542,E2 29651.542} C_VEL
LIN {X 0,Y 671.085,Z 800.857,A -85,B 0,C 180,E1 29650.746,E2 29650.746} C_VEL
LIN {X 0,Y 670.016,Z 829.873,A -85,B 0,C 180,E1 29650.195,E2 29650.195} C_VEL
LIN {X 0,Y 668.778,Z 854.868,A -85,B 0,C 180,E1 29649.555,E2 29649.555} C_VEL
LIN {X 0,Y 667.54,Z 876.53,A -85,B 0,C 180,E1 29648.875,E2 29648.875} C_VEL
LIN {X 0,Y 666.266,Z 897.129,A -85,B 0,C 180,E1 29648.114,E2 29648.114} C_VEL
LIN {X 0,Y 664.868,Z 917.41,A -85,B 0,C 180,E1 29647.252,E2 29647.252} C_VEL
LIN {X 0,Y 663.005,Z 942.493,A -85,B 0,C 180,E1 29646.028,E2 29646.028} C_VEL
LIN {X 0,Y 660.995,Z 967.064,A -85,B 0,C 180,E1 29644.622,E2 29644.622} C_VEL
LIN {X 0,Y 659.208,Z 988.805,A -85,B 0,C 180,E1 29643.201,E2 29643.201} C_VEL
LIN {X 0,Y 657.361,Z 1011.161,A -85,B 0,C 180,E1 29641.551,E2 29641.551} C_VEL
LIN {X 0,Y 655.479,Z 1033.532,A -85,B 0,C 180,E1 29639.671,E2 29639.671} C_VEL
LIN {X 0,Y 653.905,Z 1053.431,A -85,B 0,C 180,E1 29637.774,E2 29637.774} C_VEL
LIN {X 0,Y 652.47,Z 1071.873,A -85,B 0,C 180,E1 29635.8,E2 29635.8} C_VEL
LIN {X 0,Y 651.226,Z 1089.764,A -85,B 0,C 180,E1 29633.625,E2 29633.625} C_VEL
LIN {X 0,Y 650.36,Z 1103.488,A -85,B 0,C 180,E1 29631.749,E2 29631.749} C_VEL
LIN {X 0,Y 649.692,Z 1115.123,A -85,B 0,C 180,E1 29629.979,E2 29629.979} C_VEL
LIN {X 0,Y 649.171,Z 1125.516,A -85,B 0,C 180,E1 29628.221,E2 29628.221} C_VEL
LIN {X 0,Y 648.719,Z 1136.144,A -85,B 0,C 180,E1 29626.2,E2 29626.2} C_VEL
LIN {X 0,Y 648.339,Z 1147.185,A -85,B 0,C 180,E1 29623.74,E2 29623.74} C_VEL
LIN {X 0,Y 648.136,Z 1155.346,A -85,B 0,C 180,E1 29621.57,E2 29621.57} C_VEL
LIN {X 0,Y 648.014,Z 1161.98,A -85,B 0,C 180,E1 29619.414,E2 29619.414} C_VEL
LIN {X 0,Y 647.95,Z 1167.41,A -85,B 0,C 180,E1 29617.181,E2 29617.181} C_VEL
LIN {X 0,Y 647.919,Z 1171.498,A -85,B 0,C 180,E1 29614.87,E2 29614.87} C_VEL
LIN {X 0,Y 647.908,Z 1174.059,A -85,B 0,C 180,E1 29612.478,E2 29612.478} C_VEL
LIN {X 0,Y 647.902,Z 1174.954,A -85,B 0,C 180,E1 29610.178,E2 29610.178} C_VEL
LIN {X 0,Y 647.912,Z 1174.286,A -85,B 0,C 180,E1 29607.79,E2 29607.79} C_VEL
LIN {X 0,Y 647.913,Z 1172.108,A -85,B 0,C 180,E1 29605.487,E2 29605.487} C_VEL
LIN {X 0,Y 647.937,Z 1168.003,A -85,B 0,C 180,E1 29602.999,E2 29602.999} C_VEL
LIN {X 0,Y 647.998,Z 1162.725,A -85,B 0,C 180,E1 29600.767,E2 29600.767} C_VEL
LIN {X 0,Y 648.124,Z 1155.953,A -85,B 0,C 180,E1 29598.522,E2 29598.522} C_VEL
LIN {X 0,Y 648.308,Z 1148.262,A -85,B 0,C 180,E1 29596.443,E2 29596.443} C_VEL
LIN {X 0,Y 648.666,Z 1137.986,A -85,B 0,C 180,E1 29594.076,E2 29594.076} C_VEL
LIN {X 0,Y 649.15,Z 1126.03,A -85,B 0,C 180,E1 29591.78,E2 29591.78} C_VEL
LIN {X 0,Y 649.659,Z 1115.696,A -85,B 0,C 180,E1 29590.022,E2 29590.022} C_VEL
LIN {X 0,Y 650.327,Z 1103.948,A -85,B 0,C 180,E1 29588.228,E2 29588.228} C_VEL
LIN {X 0,Y 651.129,Z 1091.092,A -85,B 0,C 180,E1 29586.459,E2 29586.459} C_VEL
LIN {X 0,Y 652.313,Z 1074.342,A -85,B 0,C 180,E1 29584.391,E2 29584.391} C_VEL
LIN {X 0,Y 653.828,Z 1054.443,A -85,B 0,C 180,E1 29582.238,E2 29582.238} C_VEL
LIN {X 0,Y 655.315,Z 1035.576,A -85,B 0,C 180,E1 29580.426,E2 29580.426} C_VEL
LIN {X 0,Y 657.07,Z 1014.392,A -85,B 0,C 180,E1 29578.616,E2 29578.616} C_VEL
LIN {X 0,Y 658.951,Z 992.171,A -85,B 0,C 180,E1 29576.943,E2 29576.943} C_VEL
LIN {X 0,Y 660.811,Z 969.35,A -85,B 0,C 180,E1 29575.431,E2 29575.431} C_VEL
LIN {X 0,Y 662.594,Z 947.08,A -85,B 0,C 180,E1 29574.132,E2 29574.132} C_VEL
LIN {X 0,Y 664.585,Z 921.47,A -85,B 0,C 180,E1 29572.84,E2 29572.84} C_VEL
LIN {X 0,Y 666.202,Z 898.107,A -85,B 0,C 180,E1 29571.835,E2 29571.835} C_VEL
LIN {X 0,Y 667.49,Z 877.366,A -85,B 0,C 180,E1 29571.064,E2 29571.064} C_VEL
LIN {X 0,Y 668.757,Z 855.356,A -85,B 0,C 180,E1 29570.37,E2 29570.37} C_VEL
LIN {X 0,Y 669.948,Z 831.183,A -85,B 0,C 180,E1 29569.746,E2 29569.746} C_VEL
LIN {X 0,Y 671.048,Z 802.443,A -85,B 0,C 180,E1 29569.188,E2 29569.188} C_VEL
LIN {X 0,Y 671.998,Z 750.991,A -85,B 0,C 180,E1 29568.5,E2 29568.5} C_VEL
LIN {X 0,Y 675.389,Z 527.679,A -85,B 0,C 180,E1 29565.584,E2 29565.584} C_VEL
LIN {X 0,Y 677.99,Z 365.15,A -85,B 0,C 180,E1 29563.399,E2 29563.399} C_VEL
LIN {X 0,Y 667.268,Z 349.346,A -85,B 0,C 180,E1 29562.169,E2 29562.169} C_VEL
LIN {X 0,Y 662.524,Z 343.095,A -85,B 0,C 180,E1 29561.61,E2 29561.61} C_VEL
LIN {X 0,Y 658.621,Z 339.052,A -85,B 0,C 180,E1 29561.157,E2 29561.157} C_VEL
LIN {X 0,Y 655.357,Z 336.113,A -85,B 0,C 180,E1 29560.769,E2 29560.769} C_VEL
LIN {X 0,Y 654.337,Z 333.61,A -85,B 0,C 180,E1 29560.27,E2 29560.27} C_VEL
LIN {X 0,Y 652.095,Z 330.082,A -85,B 0,C 180,E1 29559.396,E2 29559.396} C_VEL
LIN {X 0,Y 651.296,Z 328.333,A -85,B 0,C 180,E1 29559.009,E2 29559.009} C_VEL
LIN {X 0,Y 649.338,Z 325.586,A -85,B 0,C 180,E1 29558.245,E2 29558.245} C_VEL
LIN {X 0,Y 648.775,Z 323.419,A -85,B 0,C 180,E1 29557.797,E2 29557.797} C_VEL
LIN {X 0,Y 648.763,Z 323.398,A -85,B 0,C 180,E1 29554.553,E2 29554.553} C_VEL
LIN {X 0,Y 648.776,Z 323.42,A -85,B 0,C 180,E1 29551.291,E2 29551.291} C_VEL
LIN {X 0,Y 648.742,Z 323.398,A -85,B 0,C 180,E1 29548.241,E2 29548.241} C_VEL
LIN {X 0,Y 648.764,Z 323.388,A -85,B 0,C 180,E1 29545.175,E2 29545.175} C_VEL
LIN {X 0,Y 648.742,Z 323.423,A -85,B 0,C 180,E1 29542.091,E2 29542.091} C_VEL
LIN {X 0,Y 648.77,Z 323.401,A -85,B 0,C 180,E1 29539.071,E2 29539.071} C_VEL
LIN {X 0,Y 648.758,Z 323.387,A -85,B 0,C 180,E1 29535.831,E2 29535.831} C_VEL
LIN {X 0,Y 648.77,Z 323.416,A -85,B 0,C 180,E1 29532.642,E2 29532.642} C_VEL
LIN {X 0,Y 648.748,Z 323.405,A -85,B 0,C 180,E1 29529.582,E2 29529.582} C_VEL
LIN {X 0,Y 648.766,Z 323.385,A -85,B 0,C 180,E1 29526.371,E2 29526.371} C_VEL
LIN {X 0,Y 648.741,Z 323.419,A -85,B 0,C 180,E1 29523.358,E2 29523.358} C_VEL
LIN {X 0,Y 648.757,Z 323.404,A -85,B 0,C 180,E1 29520.353,E2 29520.353} C_VEL
LIN {X 0,Y 648.745,Z 323.386,A -85,B 0,C 180,E1 29517.261,E2 29517.261} C_VEL
LIN {X 0,Y 648.762,Z 323.398,A -85,B 0,C 180,E1 29514.162,E2 29514.162} C_VEL
LIN {X 0,Y 648.766,Z 323.42,A -85,B 0,C 180,E1 29511.045,E2 29511.045} C_VEL
LIN {X 0,Y 648.765,Z 323.447,A -85,B 0,C 180,E1 29510.463,E2 29510.463} C_VEL
LIN {X 0,Y 650.133,Z 326.984,A -85,B 0,C 180,E1 29509.723,E2 29509.723} C_VEL
LIN {X 0,Y 651.853,Z 329.068,A -85,B 0,C 180,E1 29509.125,E2 29509.125} C_VEL
LIN {X 0,Y 653.58,Z 332.701,A -85,B 0,C 180,E1 29508.349,E2 29508.349} C_VEL
LIN {X 0,Y 654.821,Z 334.348,A -85,B 0,C 180,E1 29507.925,E2 29507.925} C_VEL
LIN {X 0,Y 656.672,Z 338.08,A -85,B 0,C 180,E1 29507.155,E2 29507.155} C_VEL
LIN {X 0,Y 657.864,Z 339.97,A -85,B 0,C 180,E1 29506.732,E2 29506.732} C_VEL
LIN {X 0,Y 660.606,Z 344.94,A -85,B 0,C 180,E1 29505.717,E2 29505.717} C_VEL
LIN {X 0,Y 663.621,Z 350.633,A -85,B 0,C 180,E1 29504.622,E2 29504.622} C_VEL
LIN {X 0,Y 668.315,Z 359.195,A -85,B 0,C 180,E1 29503.037,E2 29503.037} C_VEL
LIN {X 0,Y 675.415,Z 373.048,A -85,B 0,C 180,E1 29500.723,E2 29500.723} C_VEL
LIN {X 0,Y 678.312,Z 379.306,A -85,B 0,C 180,E1 29499.777,E2 29499.777} C_VEL
LIN {X 0,Y 675.904,Z 412.011,A -85,B 0,C 180,E1 29497.16,E2 29497.16} C_VEL
LIN {X 0,Y 673.378,Z 448.287,A -85,B 0,C 180,E1 29494.399,E2 29494.399} C_VEL
LIN {X 0,Y 670.808,Z 487.982,A -85,B 0,C 180,E1 29491.511,E2 29491.511} C_VEL
LIN {X 0,Y 668.307,Z 529.383,A -85,B 0,C 180,E1 29488.623,E2 29488.623} C_VEL
LIN {X 0,Y 667.225,Z 555.998,A -85,B 0,C 180,E1 29486.788,E2 29486.788} C_VEL
LIN {X 0,Y 668.336,Z 569.959,A -85,B 0,C 180,E1 29485.717,E2 29485.717} C_VEL
LIN {X 0,Y 671.102,Z 581.912,A -85,B 0,C 180,E1 29484.683,E2 29484.683} C_VEL
LIN {X 0,Y 675.363,Z 592.13,A -85,B 0,C 180,E1 29483.686,E2 29483.686} C_VEL
LIN {X 0,Y 681.24,Z 601.136,A -85,B 0,C 180,E1 29482.686,E2 29482.686} C_VEL
LIN {X 0,Y 688.789,Z 608.828,A -85,B 0,C 180,E1 29481.694,E2 29481.694} C_VEL
LIN {X 0,Y 698.028,Z 615.165,A -85,B 0,C 180,E1 29480.717,E2 29480.717} C_VEL
LIN {X 0,Y 706.765,Z 619.078,A -85,B 0,C 180,E1 29479.931,E2 29479.931} C_VEL
LIN {X 0,Y 710.135,Z 619.705,A -85,B 0,C 180,E1 29479.526,E2 29479.526} C_VEL
LIN {X 0,Y 712.681,Z 619.28,A -85,B 0,C 180,E1 29479.065,E2 29479.065} C_VEL
LIN {X 0,Y 714.011,Z 617.978,A -85,B 0,C 180,E1 29478.625,E2 29478.625} C_VEL
LIN {X 0,Y 714.243,Z 615.508,A -85,B 0,C 180,E1 29478.136,E2 29478.136} C_VEL
LIN {X 0,Y 713.014,Z 612.086,A -85,B 0,C 180,E1 29477.677,E2 29477.677} C_VEL
LIN {X 0,Y 710.325,Z 607.87,A -85,B 0,C 180,E1 29477.287,E2 29477.287} C_VEL
LIN {X 0,Y 702.583,Z 597.61,A -85,B 0,C 180,E1 29476.682,E2 29476.682} C_VEL
LIN {X 0,Y 695.432,Z 585.605,A -85,B 0,C 180,E1 29476.124,E2 29476.124} C_VEL
LIN {X 0,Y 689.331,Z 572.14,A -85,B 0,C 180,E1 29475.635,E2 29475.635} C_VEL
LIN {X 0,Y 684.434,Z 557.512,A -85,B 0,C 180,E1 29475.232,E2 29475.232} C_VEL
LIN {X 0,Y 680.761,Z 541.781,A -85,B 0,C 180,E1 29474.925,E2 29474.925} C_VEL
LIN {X 0,Y 679.768,Z 536.631,A -85,B 0,C 180,E1 29474.841,E2 29474.841} C_VEL
LIN {X 0,Y 677.24,Z 547.006,A -85,B 0,C 180,E1 29474.625,E2 29474.625} C_VEL
LIN {X 0,Y 675.968,Z 549.478,A -85,B 0,C 180,E1 29474.516,E2 29474.516} C_VEL
LIN {X 0,Y 675.513,Z 549.884,A -85,B 0,C 180,E1 29474.474,E2 29474.474} C_VEL
LIN {X 0,Y 672.111,Z 772.532,A -85,B 0,C 180,E1 29471.564,E2 29471.564} C_VEL
LIN {X 0,Y 671.076,Z 831.335,A -85,B 0,C 180,E1 29470.784,E2 29470.784} C_VEL
LIN {X 0,Y 670.078,Z 858.078,A -85,B 0,C 180,E1 29470.279,E2 29470.279} C_VEL
LIN {X 0,Y 668.829,Z 884.438,A -85,B 0,C 180,E1 29469.615,E2 29469.615} C_VEL
LIN {X 0,Y 667.377,Z 910.098,A -85,B 0,C 180,E1 29468.801,E2 29468.801} C_VEL
LIN {X 0,Y 665.57,Z 937.395,A -85,B 0,C 180,E1 29467.746,E2 29467.746} C_VEL
LIN {X 0,Y 663.793,Z 961.774,A -85,B 0,C 180,E1 29466.618,E2 29466.618} C_VEL
LIN {X 0,Y 661.961,Z 985.632,A -85,B 0,C 180,E1 29465.345,E2 29465.345} C_VEL
LIN {X 0,Y 659.983,Z 1009.475,A -85,B 0,C 180,E1 29463.877,E2 29463.877} C_VEL
LIN {X 0,Y 658.23,Z 1030.309,A -85,B 0,C 180,E1 29462.425,E2 29462.425} C_VEL
LIN {X 0,Y 656.424,Z 1052.406,A -85,B 0,C 180,E1 29460.681,E2 29460.681} C_VEL
LIN {X 0,Y 654.641,Z 1073.959,A -85,B 0,C 180,E1 29458.75,E2 29458.75} C_VEL
LIN {X 0,Y 653.113,Z 1093.742,A -85,B 0,C 180,E1 29456.749,E2 29456.749} C_VEL
LIN {X 0,Y 651.865,Z 1110.29,A -85,B 0,C 180,E1 29454.851,E2 29454.851} C_VEL
LIN {X 0,Y 650.915,Z 1124.467,A -85,B 0,C 180,E1 29453.052,E2 29453.052} C_VEL
LIN {X 0,Y 649.956,Z 1140.771,A -85,B 0,C 180,E1 29450.72,E2 29450.72} C_VEL
LIN {X 0,Y 649.239,Z 1154.258,A -85,B 0,C 180,E1 29448.496,E2 29448.496} C_VEL
LIN {X 0,Y 648.755,Z 1165.023,A -85,B 0,C 180,E1 29446.473,E2 29446.473} C_VEL
LIN {X 0,Y 648.378,Z 1176.07,A -85,B 0,C 180,E1 29444.067,E2 29444.067} C_VEL
LIN {X 0,Y 648.137,Z 1185.216,A -85,B 0,C 180,E1 29441.658,E2 29441.658} C_VEL
LIN {X 0,Y 648.001,Z 1192.634,A -85,B 0,C 180,E1 29439.233,E2 29439.233} C_VEL
LIN {X 0,Y 647.937,Z 1198.088,A -85,B 0,C 180,E1 29436.912,E2 29436.912} C_VEL
LIN {X 0,Y 647.912,Z 1201.915,A -85,B 0,C 180,E1 29434.602,E2 29434.602} C_VEL
LIN {X 0,Y 647.91,Z 1204.207,A -85,B 0,C 180,E1 29432.298,E2 29432.298} C_VEL
LIN {X 0,Y 647.902,Z 1204.969,A -85,B 0,C 180,E1 29429.822,E2 29429.822} C_VEL
LIN {X 0,Y 647.908,Z 1204.094,A -85,B 0,C 180,E1 29427.522,E2 29427.522} C_VEL
LIN {X 0,Y 647.915,Z 1201.665,A -85,B 0,C 180,E1 29425.219,E2 29425.219} C_VEL
LIN {X 0,Y 647.948,Z 1197.633,A -85,B 0,C 180,E1 29422.866,E2 29422.866} C_VEL
LIN {X 0,Y 648.015,Z 1191.896,A -85,B 0,C 180,E1 29420.496,E2 29420.496} C_VEL
LIN {X 0,Y 648.143,Z 1184.592,A -85,B 0,C 180,E1 29418.159,E2 29418.159} C_VEL
LIN {X 0,Y 648.411,Z 1175.143,A -85,B 0,C 180,E1 29415.715,E2 29415.715} C_VEL
LIN {X 0,Y 648.772,Z 1164.546,A -85,B 0,C 180,E1 29413.433,E2 29413.433} C_VEL
LIN {X 0,Y 649.265,Z 1153.722,A -85,B 0,C 180,E1 29411.41,E2 29411.41} C_VEL
LIN {X 0,Y 649.989,Z 1140.15,A -85,B 0,C 180,E1 29409.184,E2 29409.184} C_VEL
LIN {X 0,Y 650.92,Z 1124.398,A -85,B 0,C 180,E1 29406.938,E2 29406.938} C_VEL
LIN {X 0,Y 651.868,Z 1110.271,A -85,B 0,C 180,E1 29405.147,E2 29405.147} C_VEL
LIN {X 0,Y 653.175,Z 1092.843,A -85,B 0,C 180,E1 29403.153,E2 29403.153} C_VEL
LIN {X 0,Y 654.709,Z 1073.195,A -85,B 0,C 180,E1 29401.178,E2 29401.178} C_VEL
LIN {X 0,Y 656.47,Z 1051.793,A -85,B 0,C 180,E1 29399.268,E2 29399.268} C_VEL
LIN {X 0,Y 658.232,Z 1030.277,A -85,B 0,C 180,E1 29397.572,E2 29397.572} C_VEL
LIN {X 0,Y 660.064,Z 1008.625,A -85,B 0,C 180,E1 29396.067,E2 29396.067} C_VEL
LIN {X 0,Y 662.033,Z 984.743,A -85,B 0,C 180,E1 29394.604,E2 29394.604} C_VEL
LIN {X 0,Y 663.864,Z 960.728,A -85,B 0,C 180,E1 29393.33,E2 29393.33} C_VEL
LIN {X 0,Y 665.666,Z 936.006,A -85,B 0,C 180,E1 29392.195,E2 29392.195} C_VEL
LIN {X 0,Y 667.417,Z 909.343,A -85,B 0,C 180,E1 29391.173,E2 29391.173} C_VEL
LIN {X 0,Y 668.866,Z 883.729,A -85,B 0,C 180,E1 29390.364,E2 29390.364} C_VEL
LIN {X 0,Y 670.115,Z 857.284,A -85,B 0,C 180,E1 29389.704,E2 29389.704} C_VEL
LIN {X 0,Y 671.11,Z 830.11,A -85,B 0,C 180,E1 29389.197,E2 29389.197} C_VEL
LIN {X 0,Y 672.49,Z 747.16,A -85,B 0,C 180,E1 29388.109,E2 29388.109} C_VEL
LIN {X 0,Y 675.913,Z 529.232,A -85,B 0,C 180,E1 29385.246,E2 29385.246} C_VEL
LIN {X 0,Y 678.564,Z 514.714,A -85,B 0,C 180,E1 29384.913,E2 29384.913} C_VEL
LIN {X 0,Y 682.722,Z 486.657,A -85,B 0,C 180,E1 29384.485,E2 29384.485} C_VEL
LIN {X 0,Y 685.639,Z 465.444,A -85,B 0,C 180,E1 29384.233,E2 29384.233} C_VEL
LIN {X 0,Y 687.606,Z 454.208,A -85,B 0,C 180,E1 29383.942,E2 29383.942} C_VEL
LIN {X 0,Y 691.103,Z 430.183,A -85,B 0,C 180,E1 29383.562,E2 29383.562} C_VEL
LIN {X 0,Y 695.614,Z 397.314,A -85,B 0,C 180,E1 29383.209,E2 29383.209} C_VEL
LIN {X 0,Y 697.113,Z 387.882,A -85,B 0,C 180,E1 29382.937,E2 29382.937} C_VEL
LIN {X 0,Y 698.776,Z 376.159,A -85,B 0,C 180,E1 29382.708,E2 29382.708} C_VEL
LIN {X 0,Y 698.06,Z 376.384,A -85,B 0,C 180,E1 29382.206,E2 29382.206} C_VEL
LIN {X 0,Y 695.879,Z 375.867,A -85,B 0,C 180,E1 29381.703,E2 29381.703} C_VEL
LIN {X 0,Y 692.306,Z 374.542,A -85,B 0,C 180,E1 29381.248,E2 29381.248} C_VEL
LIN {X 0,Y 684.897,Z 370.354,A -85,B 0,C 180,E1 29380.489,E2 29380.489} C_VEL
LIN {X 0,Y 675.604,Z 361.677,A -85,B 0,C 180,E1 29379.414,E2 29379.414} C_VEL
LIN {X 0,Y 664.046,Z 345.465,A -85,B 0,C 180,E1 29377.864,E2 29377.864} C_VEL
LIN {X 0,Y 656.749,Z 335.339,A -85,B 0,C 180,E1 29376.833,E2 29376.833} C_VEL
LIN {X 0,Y 653.29,Z 330.844,A -85,B 0,C 180,E1 29376.336,E2 29376.336} C_VEL
LIN {X 0,Y 652.246,Z 329.039,A -85,B 0,C 180,E1 29376.172,E2 29376.172} C_VEL
LIN {X 0,Y 649.724,Z 326.365,A -85,B 0,C 180,E1 29375.816,E2 29375.816} C_VEL
LIN {X 0,Y 648.728,Z 323.38,A -85,B 0,C 180,E1 29375.605,E2 29375.605} C_VEL
LIN {X 0,Y 648.752,Z 323.388,A -85,B 0,C 180,E1 29372.646,E2 29372.646} C_VEL
LIN {X 0,Y 648.744,Z 323.408,A -85,B 0,C 180,E1 29369.625,E2 29369.625} C_VEL
LIN {X 0,Y 648.743,Z 323.386,A -85,B 0,C 180,E1 29366.747,E2 29366.747} C_VEL
LIN {X 0,Y 648.767,Z 323.406,A -85,B 0,C 180,E1 29363.527,E2 29363.527} C_VEL
LIN {X 0,Y 648.759,Z 323.409,A -85,B 0,C 180,E1 29360.434,E2 29360.434} C_VEL
LIN {X 0,Y 648.762,Z 323.408,A -85,B 0,C 180,E1 29357.213,E2 29357.213} C_VEL
LIN {X 0,Y 648.772,Z 323.42,A -85,B 0,C 180,E1 29354.094,E2 29354.094} C_VEL
LIN {X 0,Y 648.737,Z 323.439,A -85,B 0,C 180,E1 29352.658,E2 29352.658} C_VEL
LIN {X 0,Y 651.413,Z 333.32,A -85,B 0,C 180,E1 29352.252,E2 29352.252} C_VEL
LIN {X 0,Y 651.464,Z 405.78,A -85,B 0,C 180,E1 29349.765,E2 29349.765} C_VEL
LIN {X 0,Y 651.827,Z 483.936,A -85,B 0,C 180,E1 29346.961,E2 29346.961} C_VEL
LIN {X 0,Y 652.048,Z 550.737,A -85,B 0,C 180,E1 29344.486,E2 29344.486} C_VEL
LIN {X 0,Y 651.874,Z 627.279,A -85,B 0,C 180,E1 29341.582,E2 29341.582} C_VEL
LIN {X 0,Y 651.326,Z 707.853,A -85,B 0,C 180,E1 29338.461,E2 29338.461} C_VEL
LIN {X 0,Y 650.659,Z 784.044,A -85,B 0,C 180,E1 29335.461,E2 29335.461} C_VEL
LIN {X 0,Y 650.003,Z 843.52,A -85,B 0,C 180,E1 29333.109,E2 29333.109} C_VEL
LIN {X 0,Y 649.548,Z 959.656,A -85,B 0,C 180,E1 29331.766,E2 29331.766} C_VEL
LIN {X 0,Y 649.517,Z 971.868,A -85,B 0,C 180,E1 29331.51,E2 29331.51} C_VEL
LIN {X 0,Y 649.465,Z 982.526,A -85,B 0,C 180,E1 29331.188,E2 29331.188} C_VEL
LIN {X 0,Y 649.374,Z 993.526,A -85,B 0,C 180,E1 29330.751,E2 29330.751} C_VEL
LIN {X 0,Y 649.227,Z 1005.174,A -85,B 0,C 180,E1 29330.157,E2 29330.157} C_VEL
LIN {X 0,Y 649.043,Z 1017.936,A -85,B 0,C 180,E1 29329.302,E2 29329.302} C_VEL
LIN {X 0,Y 648.881,Z 1026.976,A -85,B 0,C 180,E1 29328.534,E2 29328.534} C_VEL
LIN {X 0,Y 648.735,Z 1034.842,A -85,B 0,C 180,E1 29327.719,E2 29327.719} C_VEL
LIN {X 0,Y 648.609,Z 1041.982,A -85,B 0,C 180,E1 29326.811,E2 29326.811} C_VEL
LIN {X 0,Y 648.494,Z 1048.811,A -85,B 0,C 180,E1 29325.718,E2 29325.718} C_VEL
LIN {X 0,Y 648.396,Z 1054.182,A -85,B 0,C 180,E1 29324.527,E2 29324.527} C_VEL
LIN {X 0,Y 648.344,Z 1057.653,A -85,B 0,C 180,E1 29323.422,E2 29323.422} C_VEL
LIN {X 0,Y 648.322,Z 1059.699,A -85,B 0,C 180,E1 29322.388,E2 29322.388} C_VEL
LIN {X 0,Y 648.3,Z 1060.67,A -85,B 0,C 180,E1 29321.261,E2 29321.261} C_VEL
LIN {X 0,Y 648.307,Z 1060.19,A -85,B 0,C 180,E1 29319.929,E2 29319.929} C_VEL
LIN {X 0,Y 648.312,Z 1058.551,A -85,B 0,C 180,E1 29318.927,E2 29318.927} C_VEL
LIN {X 0,Y 647.35,Z 1057.004,A -85,B 0,C 180,E1 29318.259,E2 29318.259} C_VEL
LIN {X 0,Y 642.995,Z 1053.468,A -85,B 0,C 180,E1 29317.063,E2 29317.063} C_VEL
LIN {X 0,Y 640.867,Z 1050.446,A -85,B 0,C 180,E1 29316.339,E2 29316.339} C_VEL
LIN {X 0,Y 640.541,Z 1048.518,A -85,B 0,C 180,E1 29315.983,E2 29315.983} C_VEL
LIN {X 0,Y 640.65,Z 1042.11,A -85,B 0,C 180,E1 29314.978,E2 29314.978} C_VEL
LIN {X 0,Y 640.782,Z 1035.09,A -85,B 0,C 180,E1 29314.092,E2 29314.092} C_VEL
LIN {X 0,Y 640.935,Z 1026.907,A -85,B 0,C 180,E1 29313.248,E2 29313.248} C_VEL
LIN {X 0,Y 641.146,Z 1016.212,A -85,B 0,C 180,E1 29312.353,E2 29312.353} C_VEL
LIN {X 0,Y 641.335,Z 1003.859,A -85,B 0,C 180,E1 29311.561,E2 29311.561} C_VEL
LIN {X 0,Y 641.486,Z 992.82,A -85,B 0,C 180,E1 29311.003,E2 29311.003} C_VEL
LIN {X 0,Y 641.588,Z 982.046,A -85,B 0,C 180,E1 29310.576,E2 29310.576} C_VEL
LIN {X 0,Y 641.674,Z 969.716,A -85,B 0,C 180,E1 29310.211,E2 29310.211} C_VEL
LIN {X 0,Y 641.719,Z 953.34,A -85,B 0,C 180,E1 29309.908,E2 29309.908} C_VEL
LIN {X 0,Y 642.19,Z 842.749,A -85,B 0,C 180,E1 29308.639,E2 29308.639} C_VEL
LIN {X 0,Y 643.081,Z 767.048,A -85,B 0,C 180,E1 29305.581,E2 29305.581} C_VEL
LIN {X 0,Y 643.995,Z 689.45,A -85,B 0,C 180,E1 29302.448,E2 29302.448} C_VEL
LIN {X 0,Y 644.904,Z 609.485,A -85,B 0,C 180,E1 29299.222,E2 29299.222} C_VEL
LIN {X 0,Y 645.592,Z 545.228,A -85,B 0,C 180,E1 29296.615,E2 29296.615} C_VEL
LIN {X 0,Y 646.832,Z 547.225,A -85,B 0,C 180,E1 29296.475,E2 29296.475} C_VEL
LIN {X 0,Y 648.61,Z 547.348,A -85,B 0,C 180,E1 29296.32,E2 29296.32} C_VEL
LIN {X 0,Y 651.344,Z 545.287,A -85,B 0,C 180,E1 29296.123,E2 29296.123} C_VEL
LIN {X 0,Y 654.927,Z 539.9,A -85,B 0,C 180,E1 29295.908,E2 29295.908} C_VEL
LIN {X 0,Y 655.147,Z 539.478,A -85,B 0,C 180,E1 29295.897,E2 29295.897} C_VEL
LIN {X 0,Y 658.589,Z 538.322,A -85,B 0,C 180,E1 29295.611,E2 29295.611} C_VEL
LIN {X 0,Y 662.399,Z 534.822,A -85,B 0,C 180,E1 29295.328,E2 29295.328} C_VEL
LIN {X 0,Y 665.819,Z 529.892,A -85,B 0,C 180,E1 29295.104,E2 29295.104} C_VEL
LIN {X 0,Y 669.67,Z 527.833,A -85,B 0,C 180,E1 29294.804,E2 29294.804} C_VEL
LIN {X 0,Y 665.93,Z 755.339,A -85,B 0,C 180,E1 29291.811,E2 29291.811} C_VEL
LIN {X 0,Y 664.962,Z 803.092,A -85,B 0,C 180,E1 29291.164,E2 29291.164} C_VEL
LIN {X 0,Y 663.776,Z 831.624,A -85,B 0,C 180,E1 29290.603,E2 29290.603} C_VEL
LIN {X 0,Y 662.519,Z 855.325,A -85,B 0,C 180,E1 29289.988,E2 29289.988} C_VEL
LIN {X 0,Y 661.22,Z 876.542,A -85,B 0,C 180,E1 29289.317,E2 29289.317} C_VEL
LIN {X 0,Y 659.878,Z 896.762,A -85,B 0,C 180,E1 29288.567,E2 29288.567} C_VEL
LIN {X 0,Y 658.358,Z 917.212,A -85,B 0,C 180,E1 29287.695,E2 29287.695} C_VEL
LIN {X 0,Y 656.424,Z 941.56,A -85,B 0,C 180,E1 29286.501,E2 29286.501} C_VEL
LIN {X 0,Y 654.156,Z 967.203,A -85,B 0,C 180,E1 29285.027,E2 29285.027} C_VEL
LIN {X 0,Y 652.223,Z 988.807,A -85,B 0,C 180,E1 29283.603,E2 29283.603} C_VEL
LIN {X 0,Y 650.246,Z 1011.175,A -85,B 0,C 180,E1 29281.937,E2 29281.937} C_VEL
LIN {X 0,Y 648.239,Z 1033.085,A -85,B 0,C 180,E1 29280.079,E2 29280.079} C_VEL
LIN {X 0,Y 646.498,Z 1053.178,A -85,B 0,C 180,E1 29278.147,E2 29278.147} C_VEL
LIN {X 0,Y 644.998,Z 1071.028,A -85,B 0,C 180,E1 29276.22,E2 29276.22} C_VEL
LIN {X 0,Y 643.622,Z 1089.126,A -85,B 0,C 180,E1 29274.009,E2 29274.009} C_VEL
LIN {X 0,Y 642.649,Z 1102.843,A -85,B 0,C 180,E1 29272.119,E2 29272.119} C_VEL
LIN {X 0,Y 641.909,Z 1114.548,A -85,B 0,C 180,E1 29270.326,E2 29270.326} C_VEL
LIN {X 0,Y 641.322,Z 1124.997,A -85,B 0,C 180,E1 29268.546,E2 29268.546} C_VEL
LIN {X 0,Y 640.847,Z 1134.864,A -85,B 0,C 180,E1 29266.663,E2 29266.663} C_VEL
LIN {X 0,Y 640.474,Z 1144.945,A -85,B 0,C 180,E1 29264.466,E2 29264.466} C_VEL
LIN {X 0,Y 640.162,Z 1154.744,A -85,B 0,C 180,E1 29261.899,E2 29261.899} C_VEL
LIN {X 0,Y 640.024,Z 1161.731,A -85,B 0,C 180,E1 29259.624,E2 29259.624} C_VEL
LIN {X 0,Y 639.951,Z 1167.018,A -85,B 0,C 180,E1 29257.452,E2 29257.452} C_VEL
LIN {X 0,Y 639.923,Z 1171.106,A -85,B 0,C 180,E1 29255.201,E2 29255.201} C_VEL
LIN {X 0,Y 639.909,Z 1173.946,A -85,B 0,C 180,E1 29252.688,E2 29252.688} C_VEL
LIN {X 0,Y 639.894,Z 1174.947,A -85,B 0,C 180,E1 29250.359,E2 29250.359} C_VEL
LIN {X 0,Y 639.913,Z 1174.38,A -85,B 0,C 180,E1 29247.942,E2 29247.942} C_VEL
LIN {X 0,Y 639.919,Z 1172.411,A -85,B 0,C 180,E1 29245.7,E2 29245.7} C_VEL
LIN {X 0,Y 639.937,Z 1168.864,A -85,B 0,C 180,E1 29243.362,E2 29243.362} C_VEL
LIN {X 0,Y 639.998,Z 1163.381,A -85,B 0,C 180,E1 29240.895,E2 29240.895} C_VEL
LIN {X 0,Y 640.119,Z 1156.848,A -85,B 0,C 180,E1 29238.65,E2 29238.65} C_VEL
LIN {X 0,Y 640.306,Z 1149.632,A -85,B 0,C 180,E1 29236.624,E2 29236.624} C_VEL
LIN {X 0,Y 640.564,Z 1141.682,A -85,B 0,C 180,E1 29234.706,E2 29234.706} C_VEL
LIN {X 0,Y 640.95,Z 1132.893,A -85,B 0,C 180,E1 29232.853,E2 29232.853} C_VEL
LIN {X 0,Y 641.484,Z 1122.37,A -85,B 0,C 180,E1 29230.895,E2 29230.895} C_VEL
LIN {X 0,Y 642.327,Z 1107.981,A -85,B 0,C 180,E1 29228.544,E2 29228.544} C_VEL
LIN {X 0,Y 643.294,Z 1093.31,A -85,B 0,C 180,E1 29226.457,E2 29226.457} C_VEL
LIN {X 0,Y 644.375,Z 1079.088,A -85,B 0,C 180,E1 29224.644,E2 29224.644} C_VEL
LIN {X 0,Y 645.777,Z 1061.449,A -85,B 0,C 180,E1 29222.624,E2 29222.624} C_VEL
LIN {X 0,Y 647.627,Z 1040.285,A -85,B 0,C 180,E1 29220.496,E2 29220.496} C_VEL
LIN {X 0,Y 649.457,Z 1019.388,A -85,B 0,C 180,E1 29218.644,E2 29218.644} C_VEL
LIN {X 0,Y 651.46,Z 997.565,A -85,B 0,C 180,E1 29216.933,E2 29216.933} C_VEL
LIN {X 0,Y 653.583,Z 974.01,A -85,B 0,C 180,E1 29215.314,E2 29215.314} C_VEL
LIN {X 0,Y 655.483,Z 951.949,A -85,B 0,C 180,E1 29213.983,E2 29213.983} C_VEL
LIN {X 0,Y 657.352,Z 929.627,A -85,B 0,C 180,E1 29212.8,E2 29212.8} C_VEL
LIN {X 0,Y 659.485,Z 902.396,A -85,B 0,C 180,E1 29211.567,E2 29211.567} C_VEL
LIN {X 0,Y 661.071,Z 878.924,A -85,B 0,C 180,E1 29210.675,E2 29210.675} C_VEL
LIN {X 0,Y 662.429,Z 857.019,A -85,B 0,C 180,E1 29209.972,E2 29209.972} C_VEL
LIN {X 0,Y 663.62,Z 834.712,A -85,B 0,C 180,E1 29209.382,E2 29209.382} C_VEL
LIN {X 0,Y 664.701,Z 809.931,A -85,B 0,C 180,E1 29208.864,E2 29208.864} C_VEL
LIN {X 0,Y 665.617,Z 775.256,A -85,B 0,C 180,E1 29208.357,E2 29208.357} C_VEL
LIN {X 0,Y 669.276,Z 550.875,A -85,B 0,C 180,E1 29205.413,E2 29205.413} C_VEL
LIN {X 0,Y 672.43,Z 368.966,A -85,B 0,C 180,E1 29202.955,E2 29202.955} C_VEL
LIN {X 0,Y 662.768,Z 354.8,A -85,B 0,C 180,E1 29201.823,E2 29201.823} C_VEL
LIN {X 0,Y 658.646,Z 349.36,A -85,B 0,C 180,E1 29201.329,E2 29201.329} C_VEL
LIN {X 0,Y 655.206,Z 345.872,A -85,B 0,C 180,E1 29200.925,E2 29200.925} C_VEL
LIN {X 0,Y 649.631,Z 340.245,A -85,B 0,C 180,E1 29200.255,E2 29200.255} C_VEL
LIN {X 0,Y 647.179,Z 336.292,A -85,B 0,C 180,E1 29199.284,E2 29199.284} C_VEL
LIN {X 0,Y 646.393,Z 334.602,A -85,B 0,C 180,E1 29198.905,E2 29198.905} C_VEL
LIN {X 0,Y 644.286,Z 331.357,A -85,B 0,C 180,E1 29198.033,E2 29198.033} C_VEL
LIN {X 0,Y 643.602,Z 329.523,A -85,B 0,C 180,E1 29197.63,E2 29197.63} C_VEL
LIN {X 0,Y 641.301,Z 326.314,A -85,B 0,C 180,E1 29196.667,E2 29196.667} C_VEL
LIN {X 0,Y 640.802,Z 324.404,A -85,B 0,C 180,E1 29196.227,E2 29196.227} C_VEL
LIN {X 0,Y 640.819,Z 324.372,A -85,B 0,C 180,E1 29193.208,E2 29193.208} C_VEL
LIN {X 0,Y 640.804,Z 324.383,A -85,B 0,C 180,E1 29190.162,E2 29190.162} C_VEL
LIN {X 0,Y 640.827,Z 324.411,A -85,B 0,C 180,E1 29187.104,E2 29187.104} C_VEL
LIN {X 0,Y 640.826,Z 324.382,A -85,B 0,C 180,E1 29183.892,E2 29183.892} C_VEL
LIN {X 0,Y 640.826,Z 324.375,A -85,B 0,C 180,E1 29180.648,E2 29180.648} C_VEL
LIN {X 0,Y 640.808,Z 324.412,A -85,B 0,C 180,E1 29177.571,E2 29177.571} C_VEL
LIN {X 0,Y 640.822,Z 324.386,A -85,B 0,C 180,E1 29174.457,E2 29174.457} C_VEL
LIN {X 0,Y 640.802,Z 324.378,A -85,B 0,C 180,E1 29171.43,E2 29171.43} C_VEL
LIN {X 0,Y 640.808,Z 324.411,A -85,B 0,C 180,E1 29168.344,E2 29168.344} C_VEL
LIN {X 0,Y 640.821,Z 324.38,A -85,B 0,C 180,E1 29165.282,E2 29165.282} C_VEL
LIN {X 0,Y 640.815,Z 324.376,A -85,B 0,C 180,E1 29162.146,E2 29162.146} C_VEL
LIN {X 0,Y 640.821,Z 324.407,A -85,B 0,C 180,E1 29159.017,E2 29159.017} C_VEL
LIN {X 0,Y 640.825,Z 324.395,A -85,B 0,C 180,E1 29155.794,E2 29155.794} C_VEL
LIN {X 0,Y 640.799,Z 324.372,A -85,B 0,C 180,E1 29152.739,E2 29152.739} C_VEL
LIN {X 0,Y 640.836,Z 324.59,A -85,B 0,C 180,E1 29151.973,E2 29151.973} C_VEL
LIN {X 0,Y 642.129,Z 327.892,A -85,B 0,C 180,E1 29151.222,E2 29151.222} C_VEL
LIN {X 0,Y 643.991,Z 330.124,A -85,B 0,C 180,E1 29150.527,E2 29150.527} C_VEL
LIN {X 0,Y 645.825,Z 333.925,A -85,B 0,C 180,E1 29149.654,E2 29149.654} C_VEL
LIN {X 0,Y 647.018,Z 335.47,A -85,B 0,C 180,E1 29149.223,E2 29149.223} C_VEL
LIN {X 0,Y 649.036,Z 339.333,A -85,B 0,C 180,E1 29148.357,E2 29148.357} C_VEL
LIN {X 0,Y 649.958,Z 340.759,A -85,B 0,C 180,E1 29148.013,E2 29148.013} C_VEL
LIN {X 0,Y 652.122,Z 344.721,A -85,B 0,C 180,E1 29147.154,E2 29147.154} C_VEL
LIN {X 0,Y 655.717,Z 351.339,A -85,B 0,C 180,E1 29145.788,E2 29145.788} C_VEL
LIN {X 0,Y 660.712,Z 360.491,A -85,B 0,C 180,E1 29144.012,E2 29144.012} C_VEL
LIN {X 0,Y 667.656,Z 373.846,A -85,B 0,C 180,E1 29141.669,E2 29141.669} C_VEL
LIN {X 0,Y 672.577,Z 384.102,A -85,B 0,C 180,E1 29140.051,E2 29140.051} C_VEL
LIN {X 0,Y 670.031,Z 416.101,A -85,B 0,C 180,E1 29137.474,E2 29137.474} C_VEL
LIN {X 0,Y 667.336,Z 451.982,A -85,B 0,C 180,E1 29134.721,E2 29134.721} C_VEL
LIN {X 0,Y 664.556,Z 491.726,A -85,B 0,C 180,E1 29131.807,E2 29131.807} C_VEL
LIN {X 0,Y 661.852,Z 533.197,A -85,B 0,C 180,E1 29128.89,E2 29128.89} C_VEL
LIN {X 0,Y 660.709,Z 559.029,A -85,B 0,C 180,E1 29127.091,E2 29127.091} C_VEL
LIN {X 0,Y 661.808,Z 573.624,A -85,B 0,C 180,E1 29125.96,E2 29125.96} C_VEL
LIN {X 0,Y 664.493,Z 585.637,A -85,B 0,C 180,E1 29124.913,E2 29124.913} C_VEL
LIN {X 0,Y 668.632,Z 596.003,A -85,B 0,C 180,E1 29123.9,E2 29123.9} C_VEL
LIN {X 0,Y 674.832,Z 605.885,A -85,B 0,C 180,E1 29122.805,E2 29122.805} C_VEL
LIN {X 0,Y 682.841,Z 614.249,A -85,B 0,C 180,E1 29121.727,E2 29121.727} C_VEL
LIN {X 0,Y 691.998,Z 620.744,A -85,B 0,C 180,E1 29120.737,E2 29120.737} C_VEL
LIN {X 0,Y 702.155,Z 625.521,A -85,B 0,C 180,E1 29119.828,E2 29119.828} C_VEL
LIN {X 0,Y 706.363,Z 626.497,A -85,B 0,C 180,E1 29119.371,E2 29119.371} C_VEL
LIN {X 0,Y 709.095,Z 626.219,A -85,B 0,C 180,E1 29118.92,E2 29118.92} C_VEL
LIN {X 0,Y 710.819,Z 624.751,A -85,B 0,C 180,E1 29118.398,E2 29118.398} C_VEL
LIN {X 0,Y 711.101,Z 622.459,A -85,B 0,C 180,E1 29117.936,E2 29117.936} C_VEL
LIN {X 0,Y 709.957,Z 619.065,A -85,B 0,C 180,E1 29117.466,E2 29117.466} C_VEL
LIN {X 0,Y 707.359,Z 614.949,A -85,B 0,C 180,E1 29117.07,E2 29117.07} C_VEL
LIN {X 0,Y 699.406,Z 604.633,A -85,B 0,C 180,E1 29116.437,E2 29116.437} C_VEL
LIN {X 0,Y 691.838,Z 592.301,A -85,B 0,C 180,E1 29115.837,E2 29115.837} C_VEL
LIN {X 0,Y 685.41,Z 578.679,A -85,B 0,C 180,E1 29115.313,E2 29115.313} C_VEL
LIN {X 0,Y 680.143,Z 563.804,A -85,B 0,C 180,E1 29114.873,E2 29114.873} C_VEL
LIN {X 0,Y 679.923,Z 563.434,A -85,B 0,C 180,E1 29114.854,E2 29114.854} C_VEL
LIN {X 0,Y 675.727,Z 599.857,A -85,B 0,C 180,E1 29114.495,E2 29114.495} C_VEL
LIN {X 0,Y 672.123,Z 622.005,A -85,B 0,C 180,E1 29114.182,E2 29114.182} C_VEL
LIN {X 0,Y 669.776,Z 631.025,A -85,B 0,C 180,E1 29113.975,E2 29113.975} C_VEL
LIN {X 0,Y 668.649,Z 632.825,A -85,B 0,C 180,E1 29113.875,E2 29113.875} C_VEL
LIN {X 0,Y 668.392,Z 633.226,A -85,B 0,C 180,E1 29113.848,E2 29113.848} C_VEL
LIN {X 0,Y 665.089,Z 828.658,A -85,B 0,C 180,E1 29111.278,E2 29111.278} C_VEL
LIN {X 0,Y 664.089,Z 855.225,A -85,B 0,C 180,E1 29110.791,E2 29110.791} C_VEL
LIN {X 0,Y 662.766,Z 881.802,A -85,B 0,C 180,E1 29110.139,E2 29110.139} C_VEL
LIN {X 0,Y 661.21,Z 907.128,A -85,B 0,C 180,E1 29109.346,E2 29109.346} C_VEL
LIN {X 0,Y 659.427,Z 933.178,A -85,B 0,C 180,E1 29108.357,E2 29108.357} C_VEL
LIN {X 0,Y 657.414,Z 958.783,A -85,B 0,C 180,E1 29107.196,E2 29107.196} C_VEL
LIN {X 0,Y 655.424,Z 983.083,A -85,B 0,C 180,E1 29105.913,E2 29105.913} C_VEL
LIN {X 0,Y 653.278,Z 1007.551,A -85,B 0,C 180,E1 29104.413,E2 29104.413} C_VEL
LIN {X 0,Y 651.271,Z 1029.492,A -85,B 0,C 180,E1 29102.88,E2 29102.88} C_VEL
LIN {X 0,Y 649.306,Z 1051.233,A -85,B 0,C 180,E1 29101.157,E2 29101.157} C_VEL
LIN {X 0,Y 647.396,Z 1072.876,A -85,B 0,C 180,E1 29099.211,E2 29099.211} C_VEL
LIN {X 0,Y 645.733,Z 1091.982,A -85,B 0,C 180,E1 29097.275,E2 29097.275} C_VEL
LIN {X 0,Y 644.302,Z 1109.925,A -85,B 0,C 180,E1 29095.209,E2 29095.209} C_VEL
LIN {X 0,Y 643.222,Z 1124.416,A -85,B 0,C 180,E1 29093.352,E2 29093.352} C_VEL
LIN {X 0,Y 642.197,Z 1140.163,A -85,B 0,C 180,E1 29091.078,E2 29091.078} C_VEL
LIN {X 0,Y 641.407,Z 1153.738,A -85,B 0,C 180,E1 29088.824,E2 29088.824} C_VEL
LIN {X 0,Y 640.866,Z 1164.56,A -85,B 0,C 180,E1 29086.775,E2 29086.775} C_VEL
LIN {X 0,Y 640.469,Z 1175.15,A -85,B 0,C 180,E1 29084.464,E2 29084.464} C_VEL
LIN {X 0,Y 640.164,Z 1184.598,A -85,B 0,C 180,E1 29081.988,E2 29081.988} C_VEL
LIN {X 0,Y 640.024,Z 1191.903,A -85,B 0,C 180,E1 29079.622,E2 29079.622} C_VEL
LIN {X 0,Y 639.955,Z 1197.531,A -85,B 0,C 180,E1 29077.269,E2 29077.269} C_VEL
LIN {X 0,Y 639.922,Z 1201.543,A -85,B 0,C 180,E1 29074.929,E2 29074.929} C_VEL
LIN {X 0,Y 639.909,Z 1204.038,A -85,B 0,C 180,E1 29072.596,E2 29072.596} C_VEL
LIN {X 0,Y 639.897,Z 1204.951,A -85,B 0,C 180,E1 29070.267,E2 29070.267} C_VEL
LIN {X 0,Y 639.911,Z 1204.262,A -85,B 0,C 180,E1 29067.76,E2 29067.76} C_VEL
LIN {X 0,Y 639.913,Z 1202.035,A -85,B 0,C 180,E1 29065.428,E2 29065.428} C_VEL
LIN {X 0,Y 639.939,Z 1198.256,A -85,B 0,C 180,E1 29063.089,E2 29063.089} C_VEL
LIN {X 0,Y 640.008,Z 1192.867,A -85,B 0,C 180,E1 29060.739,E2 29060.739} C_VEL
LIN {X 0,Y 640.153,Z 1185.515,A -85,B 0,C 180,E1 29058.283,E2 29058.283} C_VEL
LIN {X 0,Y 640.423,Z 1176.301,A -85,B 0,C 180,E1 29055.81,E2 29055.81} C_VEL
LIN {X 0,Y 640.828,Z 1165.479,A -85,B 0,C 180,E1 29053.408,E2 29053.408} C_VEL
LIN {X 0,Y 641.352,Z 1154.77,A -85,B 0,C 180,E1 29051.36,E2 29051.36} C_VEL
LIN {X 0,Y 642.128,Z 1141.361,A -85,B 0,C 180,E1 29049.108,E2 29049.108} C_VEL
LIN {X 0,Y 643.176,Z 1125.11,A -85,B 0,C 180,E1 29046.741,E2 29046.741} C_VEL
LIN {X 0,Y 644.273,Z 1110.272,A -85,B 0,C 180,E1 29044.833,E2 29044.833} C_VEL
LIN {X 0,Y 645.672,Z 1092.842,A -85,B 0,C 180,E1 29042.816,E2 29042.816} C_VEL
LIN {X 0,Y 647.354,Z 1073.358,A -85,B 0,C 180,E1 29040.835,E2 29040.835} C_VEL
LIN {X 0,Y 649.251,Z 1051.937,A -85,B 0,C 180,E1 29038.902,E2 29038.902} C_VEL
LIN {X 0,Y 651.196,Z 1030.282,A -85,B 0,C 180,E1 29037.178,E2 29037.178} C_VEL
LIN {X 0,Y 653.104,Z 1009.356,A -85,B 0,C 180,E1 29035.708,E2 29035.708} C_VEL
LIN {X 0,Y 655.133,Z 986.534,A -85,B 0,C 180,E1 29034.288,E2 29034.288} C_VEL
LIN {X 0,Y 657.105,Z 962.821,A -85,B 0,C 180,E1 29033.005,E2 29033.005} C_VEL
LIN {X 0,Y 659.018,Z 938.468,A -85,B 0,C 180,E1 29031.864,E2 29031.864} C_VEL
LIN {X 0,Y 660.964,Z 911.5,A -85,B 0,C 180,E1 29030.804,E2 29030.804} C_VEL
LIN {X 0,Y 662.546,Z 885.32,A -85,B 0,C 180,E1 29029.964,E2 29029.964} C_VEL
LIN {X 0,Y 663.915,Z 858.676,A -85,B 0,C 180,E1 29029.285,E2 29029.285} C_VEL
LIN {X 0,Y 664.983,Z 832.264,A -85,B 0,C 180,E1 29028.778,E2 29028.778} C_VEL
LIN {X 0,Y 665.964,Z 782.73,A -85,B 0,C 180,E1 29028.11,E2 29028.11} C_VEL
LIN {X 0,Y 669.28,Z 589.269,A -85,B 0,C 180,E1 29025.556,E2 29025.556} C_VEL
LIN {X 0,Y 672.471,Z 567.873,A -85,B 0,C 180,E1 29025.12,E2 29025.12} C_VEL
LIN {X 0,Y 676.933,Z 535.344,A -85,B 0,C 180,E1 29024.654,E2 29024.654} C_VEL
LIN {X 0,Y 677.673,Z 530.033,A -85,B 0,C 180,E1 29024.563,E2 29024.563} C_VEL
LIN {X 0,Y 680.111,Z 512.374,A -85,B 0,C 180,E1 29024.185,E2 29024.185} C_VEL
LIN {X 0,Y 684.15,Z 482.36,A -85,B 0,C 180,E1 29023.758,E2 29023.758} C_VEL
LIN {X 0,Y 686.176,Z 467.441,A -85,B 0,C 180,E1 29023.58,E2 29023.58} C_VEL
LIN {X 0,Y 687.744,Z 454.519,A -85,B 0,C 180,E1 29023.263,E2 29023.263} C_VEL
LIN {X 0,Y 691.031,Z 429.1,A -85,B 0,C 180,E1 29022.879,E2 29022.879} C_VEL
LIN {X 0,Y 695.138,Z 399.522,A -85,B 0,C 180,E1 29022.569,E2 29022.569} C_VEL
LIN {X 0,Y 696.191,Z 388.576,A -85,B 0,C 180,E1 29022.278,E2 29022.278} C_VEL
LIN {X 0,Y 696.599,Z 384.254,A -85,B 0,C 180,E1 29022.176,E2 29022.176} C_VEL
LIN {X 0,Y 694.278,Z 383.716,A -85,B 0,C 180,E1 29021.711,E2 29021.711} C_VEL
LIN {X 0,Y 690.181,Z 382.275,A -85,B 0,C 180,E1 29021.237,E2 29021.237} C_VEL
LIN {X 0,Y 682.438,Z 378.063,A -85,B 0,C 180,E1 29020.444,E2 29020.444} C_VEL
LIN {X 0,Y 675.884,Z 372.315,A -85,B 0,C 180,E1 29019.697,E2 29019.697} C_VEL
LIN {X 0,Y 669.429,Z 365.395,A -85,B 0,C 180,E1 29018.904,E2 29018.904} C_VEL
LIN {X 0,Y 658.113,Z 349.359,A -85,B 0,C 180,E1 29017.344,E2 29017.344} C_VEL
LIN {X 0,Y 654.847,Z 344.809,A -85,B 0,C 180,E1 29016.875,E2 29016.875} C_VEL
LIN {X 0,Y 651.617,Z 340.31,A -85,B 0,C 180,E1 29016.403,E2 29016.403} C_VEL
LIN {X 0,Y 648.179,Z 335.456,A -85,B 0,C 180,E1 29015.888,E2 29015.888} C_VEL
LIN {X 0,Y 645.367,Z 331.819,A -85,B 0,C 180,E1 29015.467,E2 29015.467} C_VEL
LIN {X 0,Y 644.412,Z 330.111,A -85,B 0,C 180,E1 29015.309,E2 29015.309} C_VEL
LIN {X 0,Y 641.873,Z 327.455,A -85,B 0,C 180,E1 29014.937,E2 29014.937} C_VEL
LIN {X 0,Y 640.828,Z 324.391,A -85,B 0,C 180,E1 29014.716,E2 29014.716} C_VEL
LIN {X 0,Y 640.809,Z 324.356,A -85,B 0,C 180,E1 29011.403,E2 29011.403} C_VEL
LIN {X 0,Y 640.838,Z 324.41,A -85,B 0,C 180,E1 29008.316,E2 29008.316} C_VEL
LIN {X 0,Y 640.797,Z 324.355,A -85,B 0,C 180,E1 29005.114,E2 29005.114} C_VEL
LIN {X 0,Y 640.829,Z 324.41,A -85,B 0,C 180,E1 29002.055,E2 29002.055} C_VEL
LIN {X 0,Y 640.795,Z 324.413,A -85,B 0,C 180,E1 28998.939,E2 28998.939} C_VEL
LIN {X 0,Y 640.834,Z 324.405,A -85,B 0,C 180,E1 28995.846,E2 28995.846} C_VEL
LIN {X 0,Y 640.823,Z 324.561,A -85,B 0,C 180,E1 28992.842,E2 28992.842} C_VEL
LIN {X 0,Y 643.737,Z 335.23,A -85,B 0,C 180,E1 28992.4,E2 28992.4} C_VEL
LIN {X 0,Y 643.792,Z 413.673,A -85,B 0,C 180,E1 28989.702,E2 28989.702} C_VEL
LIN {X 0,Y 644.233,Z 497.236,A -85,B 0,C 180,E1 28986.685,E2 28986.685} C_VEL
LIN {X 0,Y 644.343,Z 571.403,A -85,B 0,C 180,E1 28983.915,E2 28983.915} C_VEL
LIN {X 0,Y 643.959,Z 650.073,A -85,B 0,C 180,E1 28980.89,E2 28980.89} C_VEL
LIN {X 0,Y 643.539,Z 713.272,A -85,B 0,C 180,E1 28978.442,E2 28978.442} C_VEL
LIN {X 0,Y 642.838,Z 791.312,A -85,B 0,C 180,E1 28975.361,E2 28975.361} C_VEL
LIN {X 0,Y 642.116,Z 845.407,A -85,B 0,C 180,E1 28973.215,E2 28973.215} C_VEL
LIN {X 0,Y 641.68,Z 960.743,A -85,B 0,C 180,E1 28971.879,E2 28971.879} C_VEL
LIN {X 0,Y 641.656,Z 972.99,A -85,B 0,C 180,E1 28971.619,E2 28971.619} C_VEL
LIN {X 0,Y 641.601,Z 984.635,A -85,B 0,C 180,E1 28971.26,E2 28971.26} C_VEL
LIN {X 0,Y 641.498,Z 996.707,A -85,B 0,C 180,E1 28970.761,E2 28970.761} C_VEL
LIN {X 0,Y 641.313,Z 1009.886,A -85,B 0,C 180,E1 28970.034,E2 28970.034} C_VEL
LIN {X 0,Y 641.162,Z 1020.111,A -85,B 0,C 180,E1 28969.305,E2 28969.305} C_VEL
LIN {X 0,Y 641.002,Z 1028.521,A -85,B 0,C 180,E1 28968.574,E2 28968.574} C_VEL
LIN {X 0,Y 640.849,Z 1036.332,A -85,B 0,C 180,E1 28967.749,E2 28967.749} C_VEL
LIN {X 0,Y 640.714,Z 1043.423,A -85,B 0,C 180,E1 28966.83,E2 28966.83} C_VEL
LIN {X 0,Y 640.575,Z 1050.656,A -85,B 0,C 180,E1 28965.63,E2 28965.63} C_VEL
LIN {X 0,Y 640.482,Z 1055.802,A -85,B 0,C 180,E1 28964.424,E2 28964.424} C_VEL
LIN {X 0,Y 640.427,Z 1058.898,A -85,B 0,C 180,E1 28963.398,E2 28963.398} C_VEL
LIN {X 0,Y 640.402,Z 1060.866,A -85,B 0,C 180,E1 28962.368,E2 28962.368} C_VEL
LIN {X 0,Y 640.377,Z 1061.789,A -85,B 0,C 180,E1 28961.237,E2 28961.237} C_VEL
LIN {X 0,Y 640.384,Z 1061.276,A -85,B 0,C 180,E1 28959.909,E2 28959.909} C_VEL
LIN {X 0,Y 640.392,Z 1059.027,A -85,B 0,C 180,E1 28958.666,E2 28958.666} C_VEL
LIN {X 0,Y 640.43,Z 1055.873,A -85,B 0,C 180,E1 28957.607,E2 28957.607} C_VEL
LIN {X 0,Y 640.481,Z 1051.827,A -85,B 0,C 180,E1 28956.63,E2 28956.63} C_VEL
LIN {X 0,Y 640.541,Z 1048.518,A -85,B 0,C 180,E1 28955.983,E2 28955.983} C_VEL
LIN {X 0,Y 639.611,Z 1045.068,A -85,B 0,C 180,E1 28955.372,E2 28955.372} C_VEL
LIN {X 0,Y 635.371,Z 1037.979,A -85,B 0,C 180,E1 28954.29,E2 28954.29} C_VEL
LIN {X 0,Y 633.318,Z 1032.899,A -85,B 0,C 180,E1 28953.657,E2 28953.657} C_VEL
LIN {X 0,Y 633.021,Z 1029.911,A -85,B 0,C 180,E1 28953.355,E2 28953.355} C_VEL
LIN {X 0,Y 633.2,Z 1020.936,A -85,B 0,C 180,E1 28952.556,E2 28952.556} C_VEL
LIN {X 0,Y 633.361,Z 1011.004,A -85,B 0,C 180,E1 28951.834,E2 28951.834} C_VEL
LIN {X 0,Y 633.579,Z 997.753,A -85,B 0,C 180,E1 28951.072,E2 28951.072} C_VEL
LIN {X 0,Y 633.71,Z 985.246,A -85,B 0,C 180,E1 28950.541,E2 28950.541} C_VEL
LIN {X 0,Y 633.795,Z 973.113,A -85,B 0,C 180,E1 28950.157,E2 28950.157} C_VEL
LIN {X 0,Y 633.832,Z 960.85,A -85,B 0,C 180,E1 28949.89,E2 28949.89} C_VEL
LIN {X 0,Y 633.915,Z 929.69,A -85,B 0,C 180,E1 28949.509,E2 28949.509} C_VEL
LIN {X 0,Y 634.333,Z 844.149,A -85,B 0,C 180,E1 28948.515,E2 28948.515} C_VEL
LIN {X 0,Y 635.234,Z 775.459,A -85,B 0,C 180,E1 28945.729,E2 28945.729} C_VEL
LIN {X 0,Y 636.21,Z 696.681,A -85,B 0,C 180,E1 28942.531,E2 28942.531} C_VEL
LIN {X 0,Y 637.225,Z 615.206,A -85,B 0,C 180,E1 28939.216,E2 28939.216} C_VEL
LIN {X 0,Y 637.853,Z 561.635,A -85,B 0,C 180,E1 28937.033,E2 28937.033} C_VEL
LIN {X 0,Y 639.05,Z 563.595,A -85,B 0,C 180,E1 28936.893,E2 28936.893} C_VEL
LIN {X 0,Y 640.634,Z 563.797,A -85,B 0,C 180,E1 28936.75,E2 28936.75} C_VEL
LIN {X 0,Y 643.325,Z 561.868,A -85,B 0,C 180,E1 28936.547,E2 28936.547} C_VEL
LIN {X 0,Y 646.87,Z 556.712,A -85,B 0,C 180,E1 28936.325,E2 28936.325} C_VEL
LIN {X 0,Y 647.694,Z 555.413,A -85,B 0,C 180,E1 28936.276,E2 28936.276} C_VEL
LIN {X 0,Y 651.29,Z 554.155,A -85,B 0,C 180,E1 28935.996,E2 28935.996} C_VEL
LIN {X 0,Y 655.143,Z 550.729,A -85,B 0,C 180,E1 28935.729,E2 28935.729} C_VEL
LIN {X 0,Y 658.033,Z 546.662,A -85,B 0,C 180,E1 28935.533,E2 28935.533} C_VEL
LIN {X 0,Y 662.293,Z 544.098,A -85,B 0,C 180,E1 28935.197,E2 28935.197} C_VEL
LIN {X 0,Y 663.717,Z 543.004,A -85,B 0,C 180,E1 28935.089,E2 28935.089} C_VEL
LIN {X 0,Y 659.733,Z 769.379,A -85,B 0,C 180,E1 28932.092,E2 28932.092} C_VEL
LIN {X 0,Y 658.79,Z 807.078,A -85,B 0,C 180,E1 28931.559,E2 28931.559} C_VEL
LIN {X 0,Y 657.556,Z 833.666,A -85,B 0,C 180,E1 28931.011,E2 28931.011} C_VEL
LIN {X 0,Y 656.286,Z 856.027,A -85,B 0,C 180,E1 28930.422,E2 28930.422} C_VEL
LIN {X 0,Y 654.893,Z 877.273,A -85,B 0,C 180,E1 28929.744,E2 28929.744} C_VEL
LIN {X 0,Y 653.427,Z 897.832,A -85,B 0,C 180,E1 28928.971,E2 28928.971} C_VEL
LIN {X 0,Y 651.69,Z 919.611,A -85,B 0,C 180,E1 28928.027,E2 28928.027} C_VEL
LIN {X 0,Y 649.546,Z 944.308,A -85,B 0,C 180,E1 28926.786,E2 28926.786} C_VEL
LIN {X 0,Y 647.294,Z 967.985,A -85,B 0,C 180,E1 28925.4,E2 28925.4} C_VEL
LIN {X 0,Y 645.262,Z 989.003,A -85,B 0,C 180,E1 28924,E2 28924} C_VEL
LIN {X 0,Y 643.155,Z 1011.188,A -85,B 0,C 180,E1 28922.331,E2 28922.331} C_VEL
LIN {X 0,Y 641.005,Z 1033.008,A -85,B 0,C 180,E1 28920.462,E2 28920.462} C_VEL
LIN {X 0,Y 639.123,Z 1052.7,A -85,B 0,C 180,E1 28918.552,E2 28918.552} C_VEL
LIN {X 0,Y 637.547,Z 1070.405,A -85,B 0,C 180,E1 28916.625,E2 28916.625} C_VEL
LIN {X 0,Y 635.981,Z 1089.052,A -85,B 0,C 180,E1 28914.326,E2 28914.326} C_VEL
LIN {X 0,Y 634.913,Z 1102.846,A -85,B 0,C 180,E1 28912.403,E2 28912.403} C_VEL
LIN {X 0,Y 634.115,Z 1114.549,A -85,B 0,C 180,E1 28910.588,E2 28910.588} C_VEL
LIN {X 0,Y 633.473,Z 1125,A -85,B 0,C 180,E1 28908.785,E2 28908.785} C_VEL
LIN {X 0,Y 632.952,Z 1134.759,A -85,B 0,C 180,E1 28906.899,E2 28906.899} C_VEL
LIN {X 0,Y 632.538,Z 1144.946,A -85,B 0,C 180,E1 28904.651,E2 28904.651} C_VEL
LIN {X 0,Y 632.185,Z 1154.743,A -85,B 0,C 180,E1 28902.052,E2 28902.052} C_VEL
LIN {X 0,Y 632.039,Z 1161.481,A -85,B 0,C 180,E1 28899.839,E2 28899.839} C_VEL
LIN {X 0,Y 631.957,Z 1166.821,A -85,B 0,C 180,E1 28897.639,E2 28897.639} C_VEL
LIN {X 0,Y 631.922,Z 1170.811,A -85,B 0,C 180,E1 28895.449,E2 28895.449} C_VEL
LIN {X 0,Y 631.912,Z 1173.718,A -85,B 0,C 180,E1 28892.994,E2 28892.994} C_VEL
LIN {X 0,Y 631.892,Z 1174.905,A -85,B 0,C 180,E1 28890.545,E2 28890.545} C_VEL
LIN {X 0,Y 631.912,Z 1174.522,A -85,B 0,C 180,E1 28888.188,E2 28888.188} C_VEL
LIN {X 0,Y 631.918,Z 1172.806,A -85,B 0,C 180,E1 28886.009,E2 28886.009} C_VEL
LIN {X 0,Y 631.939,Z 1169.635,A -85,B 0,C 180,E1 28883.733,E2 28883.733} C_VEL
